(* CODESYS project ApatitKLK1400v5-31.project
   Company: CKA
   Title: Apatit KLK 1400
   Author: Stanislav
   Version: 0.0.0.26

Project tree, tasks and I/O mapping:
  MyController : TM241CE40T/U, Schneider Electric, order no. TM241CE40T/U, version 4.0.6.18
    application Application
      task MAST (cyclic, interval 20 ms, priority 15, watchdog 100 ms x 1) calls Alarm, Operations, Indication, FC, Encoder, LevelSensors, HMI
      task Network (cyclic, interval t#10ms, priority 31) calls nothing
      program Encoder [LD]
      global variables GVL
      program Alarm [LD]
      Symbols
      global variables PersistentVars
      program Operations [LD]
      program Indication [LD]
      program FC [LD]
      program LevelSensors [LD]
      program HMI [LD]
    DI : Digital Inputs, Schneider Electric, version 4.0.6.18
        settings: IOs Usage = 3
        input  idwDI_IDW0 : DWORD  // IDW0
        input  PositionEncoderA : BOOL  // IDW0.I0
        input  PositionEncoderB : BOOL  // IDW0.I1
        input  DKS : BOOL  // IDW0.I2
        input  FaultDKSLA : BOOL  // IDW0.I3
        input  FaultDKSLB : BOOL  // IDW0.I4
        input  FaultDKODriverDrum : BOOL  // IDW0.I5
        input  FaultDKOTensionDrum : BOOL  // IDW0.I6
        input  FaultATVA : BOOL  // IDW0.I7
        input  FaultATVB : BOOL  // IDW0.I8
        input  FrontEndPosition : BOOL  // IDW0.I9
        input  RearEndPosition : BOOL  // IDW0.I10
        input  EmergencyStop : BOOL  // IDW0.I11
        input  FaultTempDriverDrum : BOOL  // IDW0.I12
        input  FaultTempTensionDrum : BOOL  // IDW0.I13
        input  FaultTempSensorBreak : BOOL  // IDW0.I14
        input  PermissionGranted : BOOL  // IDW0.I15
        input  InputModeBeltLocal : BOOL  // IDW0.I16
        input  InputModeBeltAuto : BOOL  // IDW0.I17
        input  InputModeMoveLocal : BOOL  // IDW0.I18
        input  InputModeMoveAuto : BOOL  // IDW0.I19
        input  BeltRemoteForward : BOOL  // IDW0.I20
        input  BeltRemoteReverse : BOOL  // IDW0.I21
        input  BeltRemoteStop : BOOL  // IDW0.I22
        input  MoveRemoteForward : BOOL  // IDW0.I23
        input  ibDI_IB1 : BYTE  // IB1
    DQ : Digital Outputs, Schneider Electric, version 4.0.6.18
        output BeltRunForward : BOOL  // QW0.Q0
        output BeltRunReverse : BOOL  // QW0.Q1
        output MovingForward : BOOL  // QW0.Q2
        output MovingBackward : BOOL  // QW0.Q3
        output IndicationFrontEndPosition : BOOL  // QW0.Q4
        output IndicationRearEndPosition : BOOL  // QW0.Q5
        output StatusReady : BOOL  // QW0.Q6
        output StatusFault : BOOL  // QW0.Q7
        output IndicationModeAutoBelt : BOOL  // QW0.Q8
        output IndicationModeAutoMove : BOOL  // QW0.Q9
        output IndicationFCatSetpoint : BOOL  // QW0.Q10
        output AlarmSignalDevice : BOOL  // QW0.Q11
        output Reserve1 : BOOL  // QW0.Q12
        output Reserve2 : BOOL  // QW0.Q13
        output Reserve3 : BOOL  // QW0.Q14
        output Reserve4 : BOOL  // QW0.Q15
        output qbDQ_QB1 : BYTE  // QB1
        unmapped channels: QW0
    Counters : Counters, Schneider Electric, version 4.0.6.18
        settings: Instance name = 'HscMainDualPhase_0'; B input History = 'old=-1 new=1'; A input History = 'old=-1 new=0'; Temporary Instance name = 'HscMainDualPhase_0'
    Pulse_Generators : Pulse Generators, Schneider Electric, version 4.0.6.18
    Cartridge_1 : Cartridge, Schneider Electric, version 4.0.6.18
    Cartridge_2 : Cartridge, Schneider Electric, version 4.0.6.18
    IO_Bus : IO bus - TM3, Schneider Electric, version 4.0.6.18
      Module_1 : TM3DI16/G, Schneider Electric, order no. TM3DI16/G, version 1.0.1.4
          input  iwModule_1_IW0 : WORD  // IW0
          input  MoveRemoteBackward : BOOL  // IW0.I0
          input  MoveRemoteStop : BOOL  // IW0.I1
          input  AcknowledgmentRemoteAndLocal : BOOL  // IW0.I2
          input  BeltLocalForward : BOOL  // IW0.I3
          input  BeltLocalReverse : BOOL  // IW0.I4
          input  BeltLocalStop : BOOL  // IW0.I5
          input  MoveLocalForward : BOOL  // IW0.I6
          input  MoveLocalBackward : BOOL  // IW0.I7
          input  MoveLocalStop : BOOL  // IW0.I8
          input  BeltAutoForward : BOOL  // IW0.I9
          input  BeltAutoReverse : BOOL  // IW0.I10
          input  MoveAutoForward : BOOL  // IW0.I11
          input  MoveAutoBackward : BOOL  // IW0.I12
          input  FaultPowerSupply : BOOL  // IW0.I13
          input  FaultM1 : BOOL  // IW0.I14
          input  FaultM2M3 : BOOL  // IW0.I15
      Module_2 : TM3AI2H/G, Schneider Electric, order no. TM3AI2H/G, version 1.0.0.17
          settings: KPI Configuration.KPI Configuration[0] = 35; KPI Configuration.KPI Configuration[1] = 35; KPI Configuration.KPI Configuration[2] = 60; KPI Configuration.KPI Configuration[3] = 15; KPI Configuration.KPI Configuration[4] = 60; KPI Configuration.KPI Configuration[5] = 15; KPI Configuration.KPI Configuration[6] = 32; KPI Configuration.KPI Configuration[7] = 78; KPI Configuration.KPI Configuration[8] = 32; KPI Configuration.KPI Configuration[9] = 78
          input  iiModule_2_IW0 : INT  // IW0
          input  iiModule_2_IW1 : INT  // IW1
          input  ibModule_2_IBStatusIW0 : BYTE  // IBStatusIW0
          input  ibModule_2_IBStatusIW1 : BYTE  // IBStatusIW1
    COM_Bus : COM bus, Schneider Electric, version 4.0.6.18
      TM4ES4 : TM4ES4, Schneider Electric, order no. TM4ES4, version 1.0.0.10
          settings: IPAddress = [192, 168, 201, 103]; SubnetMask = [255, 255, 255, 0]; WebServer = FALSE; FTP Server = FALSE; SoMachine Protocol = TRUE; Modbus Server = TRUE; NetManage Protocol = TRUE; SNMP protocol = TRUE; Enable Routing = TRUE; WebVisu protocol = TRUE
    Ethernet_1 : Ethernet Network, Schneider Electric, version 4.0.6.18
        settings: IPAddress = [192, 168, 200, 101]; SubnetMask = [255, 255, 255, 0]; DeviceName = 'PLCKLK1400'; WebServer = TRUE; FTP Server = TRUE; SoMachine Protocol = TRUE; Modbus Server = TRUE; NetManage Protocol = TRUE; SNMP protocol = TRUE; WebVisu protocol = TRUE; DHCP Server Active = TRUE
      Industrial_Ethernet_Manager : Industrial Ethernet Manager, Schneider Electric, version 1.0.12.21
          settings: BinaryFileSize = 396; Dhcps Host 0.Client Mac Address = [16#0, 16#0, 16#0, 16#0, 16#0]; Dhcps Host 0.Client Device Name = 'ATV340_1'; Dhcps Host 0.Client IP Address = [192, 168, 200, 102]; Dhcps Host 0.Network Mask = [255, 255, 255, 0]; Dhcps Host 0.Default Gateway = [192, 168, 200, 101]; Dhcps Host 1.Client Mac Address = [16#0, 16#0, 16#0, 16#0, 16#0]; Dhcps Host 2.Client Mac Address = [16#0, 16#0, 16#0, 16#0, 16#0]; Dhcps Host 3.Client Mac Address = [16#0, 16#0, 16#0, 16#0, 16#0]; Dhcps Host 4.Client Mac Address = [16#0, 16#0, 16#0, 16#0, 16#0]; Dhcps Host 5.Client Mac Address = [16#0, 16#0, 16#0, 16#0, 16#0]; Dhcps Host 6.Client Mac Address = [16#0, 16#0, 16#0, 16#0, 16#0]; Dhcps Host 7.Client Mac Address = [16#0, 16#0, 16#0, 16#0, 16#0]; Dhcps Host 8.Client Mac Address = [16#0, 16#0, 16#0, 16#0, 16#0]; Dhcps Host 9.Client Mac Address = [16#0, 16#0, 16#0, 16#0, 16#0]; Dhcps Host 10.Client Mac Address = [16#0, 16#0, 16#0, 16#0, 16#0]; Dhcps Host 11.Client Mac Address = [16#0, 16#0, 16#0, 16#0, 16#0]; Dhcps Host 12.Client Mac Address = [16#0, 16#0, 16#0, 16#0, 16#0]; Dhcps Host 13.Client Mac Address = [16#0, 16#0, 16#0, 16#0, 16#0]; Dhcps Host 14.Client Mac Address = [16#0, 16#0, 16#0, 16#0, 16#0]; Dhcps Host 15.Client Mac Address = [16#0, 16#0, 16#0, 16#0, 16#0]; Dhcps Host 16.Client Mac Address = [16#0, 16#0, 16#0, 16#0, 16#0]; Dhcps Host 17.Client Mac Address = [16#0, 16#0, 16#0, 16#0, 16#0]; Dhcps Host 18.Client Mac Address = [16#0, 16#0, 16#0, 16#0, 16#0]; Dhcps Host 19.Client Mac Address = [16#0, 16#0, 16#0, 16#0, 16#0]; Dhcps Host 20.Client Mac Address = [16#0, 16#0, 16#0, 16#0, 16#0]; Dhcps Host 21.Client Mac Address = [16#0, 16#0, 16#0, 16#0, 16#0]; Dhcps Host 22.Client Mac Address = [16#0, 16#0, 16#0, 16#0, 16#0]; Dhcps Host 23.Client Mac Address = [16#0, 16#0, 16#0, 16#0, 16#0]; Dhcps Host 24.Client Mac Address = [16#0, 16#0, 16#0, 16#0, 16#0]; Dhcps Host 25.Client Mac Address = [16#0, 16#0, 16#0, 16#0, 16#0]; Dhcps Host 26.Client Mac Address = [16#0, 16#0, 16#0, 16#0, 16#0]; Dhcps Host 27.Client Mac Address = [16#0, 16#0, 16#0, 16#0, 16#0]; Dhcps Host 28.Client Mac Address = [16#0, 16#0, 16#0, 16#0, 16#0]; Dhcps Host 29.Client Mac Address = [16#0, 16#0, 16#0, 16#0, 16#0]; Dhcps Host 30.Client Mac Address = [16#0, 16#0, 16#0, 16#0, 16#0]; Dhcps Host 31.Client Mac Address = [16#0, 16#0, 16#0, 16#0, 16#0]; Dhcps Host 32.Client Mac Address = [16#0, 16#0, 16#0, 16#0, 16#0]; Dhcps Host 33.Client Mac Address = [16#0, 16#0, 16#0, 16#0, 16#0]; Dhcps Host 34.Client Mac Address = [16#0, 16#0, 16#0, 16#0, 16#0];
            Dhcps Host 35.Client Mac Address = [16#0, 16#0, 16#0, 16#0, 16#0]; Dhcps Host 36.Client Mac Address = [16#0, 16#0, 16#0, 16#0, 16#0]; Dhcps Host 37.Client Mac Address = [16#0, 16#0, 16#0, 16#0, 16#0]; Dhcps Host 38.Client Mac Address = [16#0, 16#0, 16#0, 16#0, 16#0]; Dhcps Host 39.Client Mac Address = [16#0, 16#0, 16#0, 16#0, 16#0]; Dhcps Host 40.Client Mac Address = [16#0, 16#0, 16#0, 16#0, 16#0]; Dhcps Host 41.Client Mac Address = [16#0, 16#0, 16#0, 16#0, 16#0]; Dhcps Host 42.Client Mac Address = [16#0, 16#0, 16#0, 16#0, 16#0]; Dhcps Host 43.Client Mac Address = [16#0, 16#0, 16#0, 16#0, 16#0]; Dhcps Host 44.Client Mac Address = [16#0, 16#0, 16#0, 16#0, 16#0]; Dhcps Host 45.Client Mac Address = [16#0, 16#0, 16#0, 16#0, 16#0]; Dhcps Host 46.Client Mac Address = [16#0, 16#0, 16#0, 16#0, 16#0]; Dhcps Host 47.Client Mac Address = [16#0, 16#0, 16#0, 16#0, 16#0]; Dhcps Host 48.Client Mac Address = [16#0, 16#0, 16#0, 16#0, 16#0]; Dhcps Host 49.Client Mac Address = [16#0, 16#0, 16#0, 16#0, 16#0]; Dhcps Host 50.Client Mac Address = [16#0, 16#0, 16#0, 16#0, 16#0]; Dhcps Host 51.Client Mac Address = [16#0, 16#0, 16#0, 16#0, 16#0]; Dhcps Host 52.Client Mac Address = [16#0, 16#0, 16#0, 16#0, 16#0]; Dhcps Host 53.Client Mac Address = [16#0, 16#0, 16#0, 16#0, 16#0]; Dhcps Host 54.Client Mac Address = [16#0, 16#0, 16#0, 16#0, 16#0]; Dhcps Host 55.Client Mac Address = [16#0, 16#0, 16#0, 16#0, 16#0]; Dhcps Host 56.Client Mac Address = [16#0, 16#0, 16#0, 16#0, 16#0]; Dhcps Host 57.Client Mac Address = [16#0, 16#0, 16#0, 16#0, 16#0]; Dhcps Host 58.Client Mac Address = [16#0, 16#0, 16#0, 16#0, 16#0]; Dhcps Host 59.Client Mac Address = [16#0, 16#0, 16#0, 16#0, 16#0]; Dhcps Host 60.Client Mac Address = [16#0, 16#0, 16#0, 16#0, 16#0]; Dhcps Host 61.Client Mac Address = [16#0, 16#0, 16#0, 16#0, 16#0]; Dhcps Host 62.Client Mac Address = [16#0, 16#0, 16#0, 16#0, 16#0]; Dhcps Host 63.Client Mac Address = [16#0, 16#0, 16#0, 16#0, 16#0]; Dhcps Host 64.Client Mac Address = [16#0, 16#0, 16#0, 16#0, 16#0]; Dhcps Host 65.Client Mac Address = [16#0, 16#0, 16#0, 16#0, 16#0]; Dhcps Host 66.Client Mac Address = [16#0, 16#0, 16#0, 16#0, 16#0]; Dhcps Host 67.Client Mac Address = [16#0, 16#0, 16#0, 16#0, 16#0]; Dhcps Host 68.Client Mac Address = [16#0, 16#0, 16#0, 16#0, 16#0]; Dhcps Host 69.Client Mac Address = [16#0, 16#0, 16#0, 16#0, 16#0]; Dhcps Host 70.Client Mac Address = [16#0, 16#0, 16#0, 16#0, 16#0]; Dhcps Host 71.Client Mac Address = [16#0, 16#0, 16#0, 16#0, 16#0]; Dhcps Host 72.Client Mac Address = [16#0, 16#0, 16#0, 16#0, 16#0]; Dhcps Host 73.Client Mac Address = [16#0, 16#0, 16#0, 16#0, 16#0]; Dhcps Host 74.Client Mac Address = [16#0, 16#0, 16#0, 16#0, 16#0];
            Dhcps Host 75.Client Mac Address = [16#0, 16#0, 16#0, 16#0, 16#0]; Dhcps Host 76.Client Mac Address = [16#0, 16#0, 16#0, 16#0, 16#0]; Dhcps Host 77.Client Mac Address = [16#0, 16#0, 16#0, 16#0, 16#0]; Dhcps Host 78.Client Mac Address = [16#0, 16#0, 16#0, 16#0, 16#0]; Dhcps Host 79.Client Mac Address = [16#0, 16#0, 16#0, 16#0, 16#0]; Dhcps Host 80.Client Mac Address = [16#0, 16#0, 16#0, 16#0, 16#0]; Dhcps Host 81.Client Mac Address = [16#0, 16#0, 16#0, 16#0, 16#0]; Dhcps Host 82.Client Mac Address = [16#0, 16#0, 16#0, 16#0, 16#0]; Dhcps Host 83.Client Mac Address = [16#0, 16#0, 16#0, 16#0, 16#0]; Dhcps Host 84.Client Mac Address = [16#0, 16#0, 16#0, 16#0, 16#0]; Dhcps Host 85.Client Mac Address = [16#0, 16#0, 16#0, 16#0, 16#0]; Dhcps Host 86.Client Mac Address = [16#0, 16#0, 16#0, 16#0, 16#0]; Dhcps Host 87.Client Mac Address = [16#0, 16#0, 16#0, 16#0, 16#0]; Dhcps Host 88.Client Mac Address = [16#0, 16#0, 16#0, 16#0, 16#0]; Dhcps Host 89.Client Mac Address = [16#0, 16#0, 16#0, 16#0, 16#0]; Dhcps Host 90.Client Mac Address = [16#0, 16#0, 16#0, 16#0, 16#0]; Dhcps Host 91.Client Mac Address = [16#0, 16#0, 16#0, 16#0, 16#0]; Dhcps Host 92.Client Mac Address = [16#0, 16#0, 16#0, 16#0, 16#0]; Dhcps Host 93.Client Mac Address = [16#0, 16#0, 16#0, 16#0, 16#0]; Dhcps Host 94.Client Mac Address = [16#0, 16#0, 16#0, 16#0, 16#0]; Dhcps Host 95.Client Mac Address = [16#0, 16#0, 16#0, 16#0, 16#0]; Dhcps Host 96.Client Mac Address = [16#0, 16#0, 16#0, 16#0, 16#0]; Dhcps Host 97.Client Mac Address = [16#0, 16#0, 16#0, 16#0, 16#0]; Dhcps Host 98.Client Mac Address = [16#0, 16#0, 16#0, 16#0, 16#0]; Dhcps Host 99.Client Mac Address = [16#0, 16#0, 16#0, 16#0, 16#0]; Dhcps Host 100.Client Mac Address = [16#0, 16#0, 16#0, 16#0, 16#0]; Dhcps Host 101.Client Mac Address = [16#0, 16#0, 16#0, 16#0, 16#0]; Dhcps Host 102.Client Mac Address = [16#0, 16#0, 16#0, 16#0, 16#0]; Dhcps Host 103.Client Mac Address = [16#0, 16#0, 16#0, 16#0, 16#0]; Dhcps Host 104.Client Mac Address = [16#0, 16#0, 16#0, 16#0, 16#0]; Dhcps Host 105.Client Mac Address = [16#0, 16#0, 16#0, 16#0, 16#0]; Dhcps Host 106.Client Mac Address = [16#0, 16#0, 16#0, 16#0, 16#0]; Dhcps Host 107.Client Mac Address = [16#0, 16#0, 16#0, 16#0, 16#0]; Dhcps Host 108.Client Mac Address = [16#0, 16#0, 16#0, 16#0, 16#0]; Dhcps Host 109.Client Mac Address = [16#0, 16#0, 16#0, 16#0, 16#0]; Dhcps Host 110.Client Mac Address = [16#0, 16#0, 16#0, 16#0, 16#0]; Dhcps Host 111.Client Mac Address = [16#0, 16#0, 16#0, 16#0, 16#0]; Dhcps Host 112.Client Mac Address = [16#0, 16#0, 16#0, 16#0, 16#0]; Dhcps Host 113.Client Mac Address = [16#0, 16#0, 16#0, 16#0, 16#0]; Dhcps Host 114.Client Mac Address = [16#0, 16#0, 16#0, 16#0, 16#0];
            Dhcps Host 115.Client Mac Address = [16#0, 16#0, 16#0, 16#0, 16#0]; Dhcps Host 116.Client Mac Address = [16#0, 16#0, 16#0, 16#0, 16#0]; Dhcps Host 117.Client Mac Address = [16#0, 16#0, 16#0, 16#0, 16#0]; Dhcps Host 118.Client Mac Address = [16#0, 16#0, 16#0, 16#0, 16#0]; Dhcps Host 119.Client Mac Address = [16#0, 16#0, 16#0, 16#0, 16#0]; Dhcps Host 120.Client Mac Address = [16#0, 16#0, 16#0, 16#0, 16#0]; Dhcps Host 121.Client Mac Address = [16#0, 16#0, 16#0, 16#0, 16#0]; Dhcps Host 122.Client Mac Address = [16#0, 16#0, 16#0, 16#0, 16#0]; Dhcps Host 123.Client Mac Address = [16#0, 16#0, 16#0, 16#0, 16#0]; Dhcps Host 124.Client Mac Address = [16#0, 16#0, 16#0, 16#0, 16#0]; Dhcps Host 125.Client Mac Address = [16#0, 16#0, 16#0, 16#0, 16#0]; Dhcps Host 126.Client Mac Address = [16#0, 16#0, 16#0, 16#0, 16#0]; Dhcps Host 127.Client Mac Address = [16#0, 16#0, 16#0, 16#0, 16#0]; Dhcps Host 128.Client Mac Address = [16#0, 16#0, 16#0, 16#0, 16#0]; serialized Values = 235c3cdb-0ed9-49ff-9223-9c00a6bcd6bc=0|
          unmapped channels: Global Status, Healthbit 0, Healthbit 1, Healthbit 2, Healthbit 3
        ATV340_1 : Altivar 340, Schneider Electric, order no. 340, version 1.0.12.0
            settings: Default Unit-ID = 248; IPAddress = [192, 168, 200, 102]; ATV340 channel.Channel ID = 0; ATV340 channel.Read Offset = 16#0000; ATV340 channel.Write Offset = 16#0000
            input  Statusword : WORD  // Statusword
            input  Actualspeed : WORD  // Output speed
            input  MotorCurrent : WORD  // InputWord 3
            input  MotorFrequency : WORD  // InputWord 4
            input  MotorVoltage : WORD  // InputWord 5
            input  DriveState : WORD  // InputWord 6
            input  MalfunctionCode : WORD  // InputWord 7
            input  LastError : WORD  // InputWord 8
            input  FaultNumber : WORD  // InputWord 9
            input  ActualError : WORD  // InputWord 10
            input  MotorCurrent2 : WORD  // InputWord 11
            input  StateWord : WORD  // InputWord 12
            input  ETIStateWord : WORD  // InputWord 13
            input  StatusWord2 : WORD  // InputWord 14
            output Controlword : WORD  // Control word
            output SpeedReference : WORD  // Speed reference
            unmapped channels: InputWord 15, InputWord 16, InputWord 17, InputWord 18, InputWord 19, InputWord 20, InputWord 21, InputWord 22, InputWord 23, InputWord 24, InputWord 25, InputWord 26, InputWord 27, InputWord 28, InputWord 29, InputWord 30, InputWord 31, InputWord 32, OutputWord 3, OutputWord 4, OutputWord 5, OutputWord 6, OutputWord 7, OutputWord 8, OutputWord 9, OutputWord 10, OutputWord 11, OutputWord 12, OutputWord 13, OutputWord 14, OutputWord 15, OutputWord 16, OutputWord 17, OutputWord 18, OutputWord 19, OutputWord 20, OutputWord 21, OutputWord 22, OutputWord 23, OutputWord 24,
              OutputWord 25, OutputWord 26, OutputWord 27, OutputWord 28, OutputWord 29, OutputWord 30, OutputWord 31, OutputWord 32
    Serial_Line_1 : Serial line, Schneider Electric, version 4.0.6.18
    Serial_Line_2 : Serial line, Schneider Electric, version 4.0.6.18
      Modbus_Manager : Modbus Manager, Schneider Electric, version 4.0.0.2
  text list GlobalTextList
*)

// MyController/Application/GVL
VAR_GLOBAL
	
	FlagFaultCommon 			AT %MX0.0 : BOOL;
	FaultGroupUniversal 		AT %MX0.1 : BOOL;
	FaultGroupBelt 				AT %MX0.2 : BOOL;
	FaultGroupMove 				AT %MX0.3 : BOOL;
	FlagFaultLowSpeed			AT %MX0.4 : BOOL;
	FlagFaultDKSLA				AT %MX0.5 : BOOL;
	FlagFaultDKSLB				AT %MX0.6 : BOOL;
	FlagFaultDKODriverDrum		AT %MX0.7 : BOOL;
	FlagFaultDKOTensionDrum		AT %MX1.0 : BOOL;
	FlagFaultATVA				AT %MX1.1 : BOOL;
	FlagFaultATVB				AT %MX1.2 : BOOL;
	FlagEmergencyStop			AT %MX1.3 : BOOL;
	FlagFaultTempDriverDrum		AT %MX1.4 : BOOL;
	FlagFaultTempTensionDrum	AT %MX1.5 : BOOL;
	FlagFaultTempSensorBreak	AT %MX1.6 : BOOL;	
	FlagFaultPowerSupply		AT %MX1.7 : BOOL;
	FlagFaultM1					AT %MX2.0 : BOOL;
	FlagFaultM2M3				AT %MX2.1 : BOOL;
	
	CurrentStateBeltFWD			AT %MX2.2 : BOOL;
	CurrentStateBeltREV			AT %MX2.3 : BOOL;
	CurrentStateMoveFWD			AT %MX2.4 : BOOL;
	CurrentStateMoveBWD 		AT %MX2.5 : BOOL;
	
	HMIFrontendPosition			AT %MX2.6 : BOOL;
	HMIRearendPosition			AT %MX2.7 : BOOL;
	HMIReady					AT %MX3.0 : BOOL;
		
	DKSPauseGlobal 				: TIME;
	PrestartBeltPause1 			: TIME := TIME#10S0MS;
	PrestartBeltPause2 			: TIME := TIME#30S0MS;
	PrestartBeltPause3 			: TIME := T#30S;
	PrestartMovePause 			: TIME := T#10S;
	DirectionChangeBeltPause 	: TIME := T#10S;
	DirectionChangeMovePause 	: TIME := T#10S;	

	ServicePrestartBeltPause1 			: TIME;
	ServicePrestartBeltPause2 			: TIME;
	ServicePrestartBeltPause3 			: TIME;
	ServicePrestartMovePause 			: TIME;
	ServiceDirectionChangeBeltPause 	: TIME;
	ServiceDirectionChangeMovePause 	: TIME;
	
	Level1Normal 				AT %MD11 : REAL;
	Level2Normal 				AT %MD12 : REAL;
	
	Position 					AT %MD13 : REAL;
	
	FCParameter1				AT %MW32 : WORD;
	FCParameter2				AT %MW33 : WORD;
	FCParameter3				AT %MW34 : WORD;
	FCParameter4				AT %MW35 : WORD;
	FCParameter5				AT %MW36 : WORD;
	FCParameter6				AT %MW37 : WORD;
	FCParameter7				AT %MW38 : WORD;
	FCParameter8				AT %MW39 : WORD;
	FCParameter9				AT %MW40 : WORD;
	FCParameter10				AT %MW41 : WORD;
	FCParameter11				AT %MW42 : WORD;
	FCParameter12				AT %MW43 : WORD;
	FCParameter13				AT %MW44 : WORD;
	FCParameter14				AT %MW45 : WORD;
	
	Level1Real : REAL;
	Level2Real : REAL;
		
	Level1Error : BOOL;
	Level2Error : BOOL;
	
	FaultReset: BOOL;
	
	FlagPrestartSignalBeltFWD: BOOL;
	FlagPrestartSignalBeltREV: BOOL;
	FlagPrestartSignalMoveFWD: BOOL;
	FlagPrestartSignalMoveBWD: BOOL;
	
	ModeBeltLocal: BOOL;
	ModeBeltRemote: BOOL;
	ModeBeltAuto: BOOL;
	ModeMoveLocal: BOOL;
	ModeMoveRemote: BOOL;
	ModeMoveAuto: BOOL;
	
	TagBeltRunning: BOOL;
	
	TONPrestartBeltPause1: TON;
	TONPrestartBeltPause2: TON;
	TONPrestartBeltPause3: TON;
	TONPrestartMovePause: TON;
	
	AcknowledgmentAuto 		AT %MX92.0: BOOL;
	
	Blinker: BOOL;
	DKSPauseInms: TIME;
	FaultAcknowledged: BOOL;
	
	TurnOnDKS: BOOL;
		
	TONDKSPrestartPause: TON;
	TONAlarmService1: TIME;
	TONFaultM1: TON;
	TONAlarmService2: TIME;
	TONFaultM2M3: TON;
	TONAlarmService3: TIME;
	TONMeander1: TON;
	TONAlarmService4: TIME;
	TONMeander2: TON;
	TONAlarmService5: TIME;
	
	TONBootInputFilter: TON;
	TONDirectionChangeBelt1: TON;
	TONDirectionChangeBelt2: TON;
	TONDirectionChangeMove1: TON;
	TONDirectionChangeMove2: TON;
	
	TONOperationsService0: TIME;
	TONOperationsService1: TIME;
	TONOperationsService2: TIME;
	TONOperationsService3: TIME;
	TONOperationsService4: TIME;
	TONOperationsService5: TIME;
	TONOperationsService6: TIME;
	TONOperationsService7: TIME;
	TONOperationsService8: TIME;
	
	HSCEnable: BOOL;
	HSCPreset: BOOL;
	EncoderEnable: BOOL;
	EncoderPreset: BOOL;
	
	EncoderValueReal: REAL;

	StatusWordAsBits: WORD_AS_BIT;
END_VAR
VAR_GLOBAL CONSTANT
	AlwaysTRUE: BOOL := TRUE;
END_VAR
VAR_GLOBAL RETAIN
	EncoderValue: DINT;
	EncoderValueBackup: DINT;
	
	HMIDKSPauseGlobal 			AT %MW2 : INT;
	HMIPrestartBeltPause1 		AT %MW3 : INT;
	HMIPrestartBeltPause2 		AT %MW4 : INT;
	HMIPrestartBeltPause3 		AT %MW5 : INT;
	HMIPrestartMovePause 		AT %MW6 : INT;
	HMIDirectionChangeBeltPause AT %MW7 : INT;
	HMIDirectionChangeMovePause AT %MW8 : INT;
	
	SpeedLocal 					AT %MW9 : INT;
	SpeedASU 					AT %MW10 : INT;

	EncoderImpulseWeight 		AT %MD6 : REAL;
	Level1min 					AT %MD7 : REAL;
	Level1max 					AT %MD8 : REAL;
	Level2min 					AT %MD9 : REAL;
	Level2max 					AT %MD10 : REAL;
	
	PositionFront 				AT %MD14 : DINT;
	PositionEnd 				AT %MD15 : DINT;
	
	LowSpeedLimit				AT %MD24 : REAL;
	DKSImpulseWeight			AT %MD25 : REAL;
	DKSMeasuredSpeed			AT %MD26 : REAL;
END_VAR

// MyController/Application/PersistentVars
VAR_GLOBAL PERSISTENT RETAIN
	
AlarmFrequency: TIME := T#1S;
	
END_VAR

// MyController/Application/Alarm
PROGRAM Alarm
VAR
	FlagStartCounter: BOOL;
	DKSCounterTimer: TON;
	TONAlarmService6: TIME;
	
	DKSSumImpulses: REAL;
	DKSCTU: CTU;
	DKSBuffer: REAL;
END_VAR
VAR // added by the converter: edge detectors and wires of the graphical bodies
    _w1, _w2 : BOOL;
END_VAR

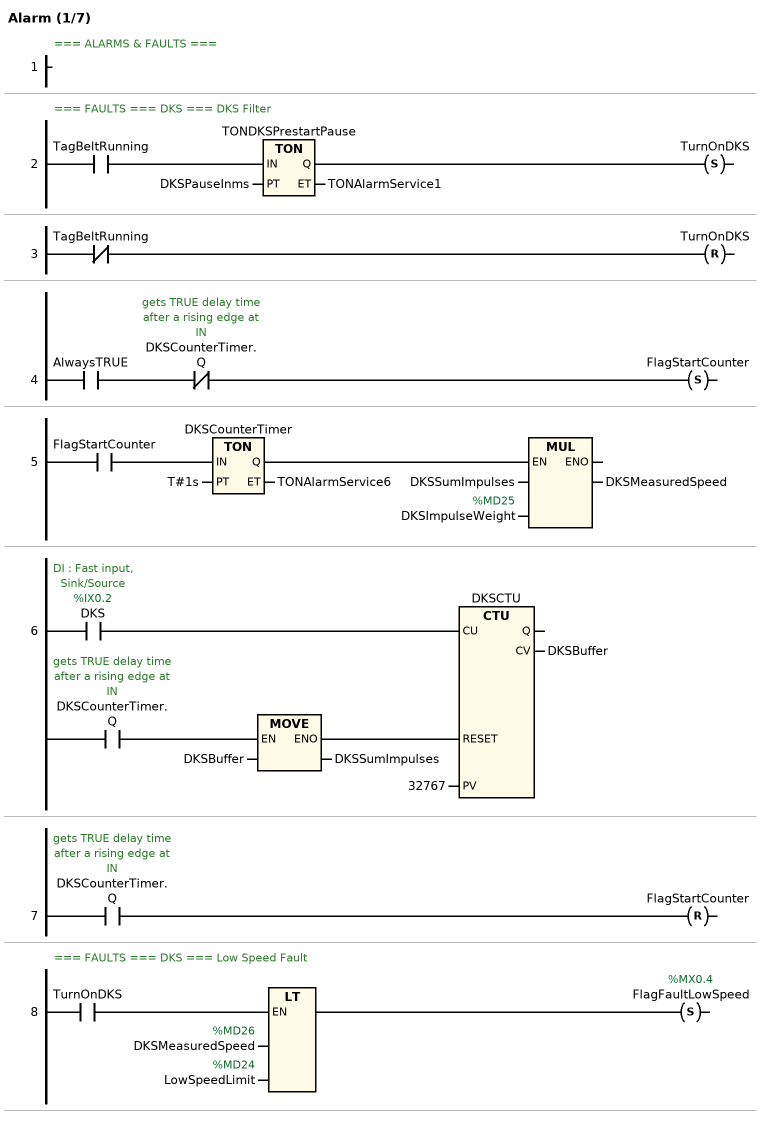
// NETWORK 1
// === ALARMS & FAULTS ===

// NETWORK 2
// === FAULTS === DKS === DKS Filter
TONDKSPrestartPause(IN := TagBeltRunning, PT := DKSPauseInms, ET => TONAlarmService1); // TON
TurnOnDKS S= TONDKSPrestartPause.Q;

// NETWORK 3
TurnOnDKS R= NOT TagBeltRunning;

// NETWORK 4
//   DKSCounterTimer.Q: gets TRUE delay time after a rising edge at IN
FlagStartCounter S= AlwaysTRUE AND NOT DKSCounterTimer.Q;

// NETWORK 5
//   DKSImpulseWeight: AT %MD25
//   DKSMeasuredSpeed: AT %MD26
DKSCounterTimer(IN := FlagStartCounter, PT := T#1s, ET => TONAlarmService6); // TON
IF DKSCounterTimer.Q THEN DKSMeasuredSpeed := DKSSumImpulses * DKSImpulseWeight; END_IF

// NETWORK 6
//   DKS: DI : Fast input, Sink/Source | AT %IX0.2
//   DKSCounterTimer.Q: gets TRUE delay time after a rising edge at IN
_w1 := DKSCounterTimer.Q;
IF _w1 THEN DKSSumImpulses := DKSBuffer; END_IF
DKSCTU(CU := DKS, RESET := _w1, PV := 32767, CV => DKSBuffer); // CTU

// NETWORK 7
//   DKSCounterTimer.Q: gets TRUE delay time after a rising edge at IN
FlagStartCounter R= DKSCounterTimer.Q;

// NETWORK 8
// === FAULTS === DKS === Low Speed Fault
//   DKSMeasuredSpeed: AT %MD26
//   LowSpeedLimit: AT %MD24
//   FlagFaultLowSpeed: AT %MX0.4
FlagFaultLowSpeed S= TurnOnDKS AND DKSMeasuredSpeed < LowSpeedLimit;

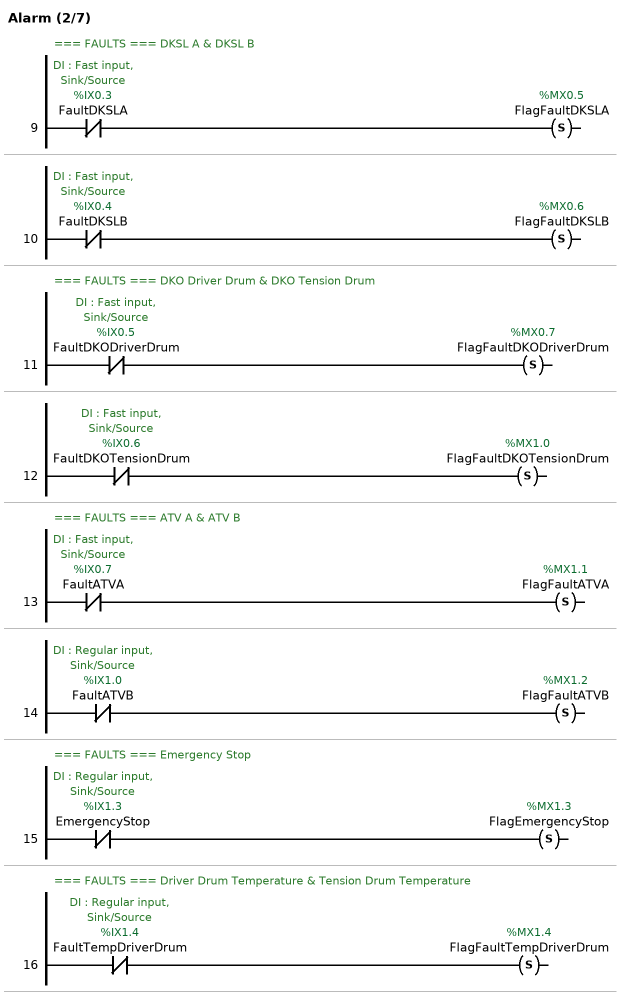
// NETWORK 9
// === FAULTS === DKSL A & DKSL B
//   FaultDKSLA: DI : Fast input, Sink/Source | AT %IX0.3
//   FlagFaultDKSLA: AT %MX0.5
FlagFaultDKSLA S= NOT FaultDKSLA;

// NETWORK 10
//   FaultDKSLB: DI : Fast input, Sink/Source | AT %IX0.4
//   FlagFaultDKSLB: AT %MX0.6
FlagFaultDKSLB S= NOT FaultDKSLB;

// NETWORK 11
// === FAULTS === DKO Driver Drum & DKO Tension Drum
//   FaultDKODriverDrum: DI : Fast input, Sink/Source | AT %IX0.5
//   FlagFaultDKODriverDrum: AT %MX0.7
FlagFaultDKODriverDrum S= NOT FaultDKODriverDrum;

// NETWORK 12
//   FaultDKOTensionDrum: DI : Fast input, Sink/Source | AT %IX0.6
//   FlagFaultDKOTensionDrum: AT %MX1.0
FlagFaultDKOTensionDrum S= NOT FaultDKOTensionDrum;

// NETWORK 13
// === FAULTS === ATV A & ATV B
//   FaultATVA: DI : Fast input, Sink/Source | AT %IX0.7
//   FlagFaultATVA: AT %MX1.1
FlagFaultATVA S= NOT FaultATVA;

// NETWORK 14
//   FaultATVB: DI : Regular input, Sink/Source | AT %IX1.0
//   FlagFaultATVB: AT %MX1.2
FlagFaultATVB S= NOT FaultATVB;

// NETWORK 15
// === FAULTS === Emergency Stop
//   EmergencyStop: DI : Regular input, Sink/Source | AT %IX1.3
//   FlagEmergencyStop: AT %MX1.3
FlagEmergencyStop S= NOT EmergencyStop;

// NETWORK 16
// === FAULTS === Driver Drum Temperature & Tension Drum Temperature
//   FaultTempDriverDrum: DI : Regular input, Sink/Source | AT %IX1.4
//   FlagFaultTempDriverDrum: AT %MX1.4
FlagFaultTempDriverDrum S= NOT FaultTempDriverDrum;

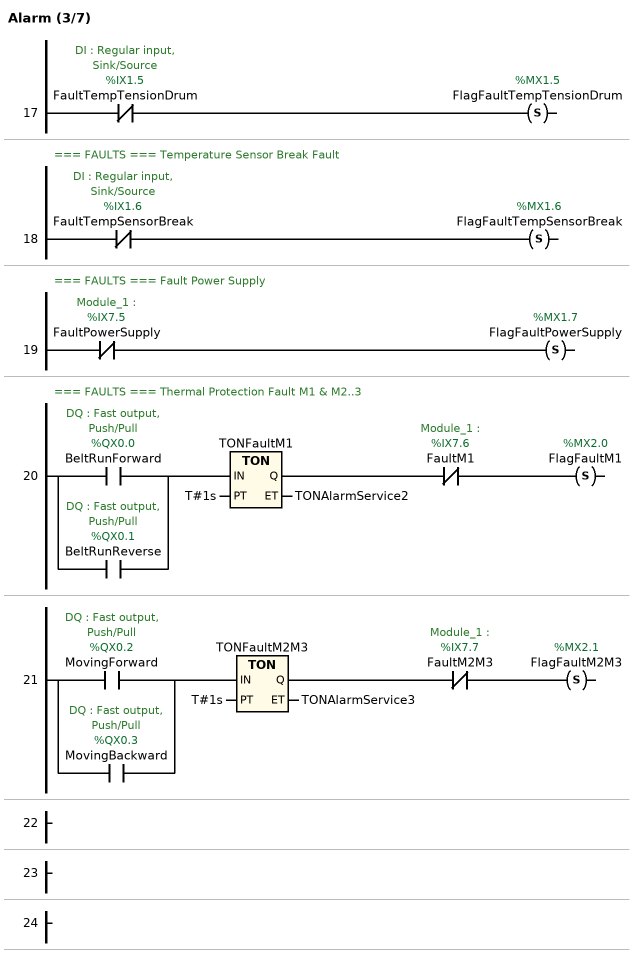
// NETWORK 17
//   FaultTempTensionDrum: DI : Regular input, Sink/Source | AT %IX1.5
//   FlagFaultTempTensionDrum: AT %MX1.5
FlagFaultTempTensionDrum S= NOT FaultTempTensionDrum;

// NETWORK 18
// === FAULTS === Temperature Sensor Break Fault
//   FaultTempSensorBreak: DI : Regular input, Sink/Source | AT %IX1.6
//   FlagFaultTempSensorBreak: AT %MX1.6
FlagFaultTempSensorBreak S= NOT FaultTempSensorBreak;

// NETWORK 19
// === FAULTS === Fault Power Supply
//   FaultPowerSupply: Module_1 : | AT %IX7.5
//   FlagFaultPowerSupply: AT %MX1.7
FlagFaultPowerSupply S= NOT FaultPowerSupply;

// NETWORK 20
// === FAULTS === Thermal Protection Fault M1 & M2..3
//   BeltRunForward: DQ : Fast output, Push/Pull | AT %QX0.0
//   BeltRunReverse: DQ : Fast output, Push/Pull | AT %QX0.1
//   FaultM1: Module_1 : | AT %IX7.6
//   FlagFaultM1: AT %MX2.0
TONFaultM1(IN := BeltRunForward OR BeltRunReverse, PT := T#1s, ET => TONAlarmService2); // TON
FlagFaultM1 S= TONFaultM1.Q AND NOT FaultM1;

// NETWORK 21
//   MovingForward: DQ : Fast output, Push/Pull | AT %QX0.2
//   MovingBackward: DQ : Fast output, Push/Pull | AT %QX0.3
//   FaultM2M3: Module_1 : | AT %IX7.7
//   FlagFaultM2M3: AT %MX2.1
TONFaultM2M3(IN := MovingForward OR MovingBackward, PT := T#1s, ET => TONAlarmService3); // TON
FlagFaultM2M3 S= TONFaultM2M3.Q AND NOT FaultM2M3;

// NETWORK 22

// NETWORK 23

// NETWORK 24

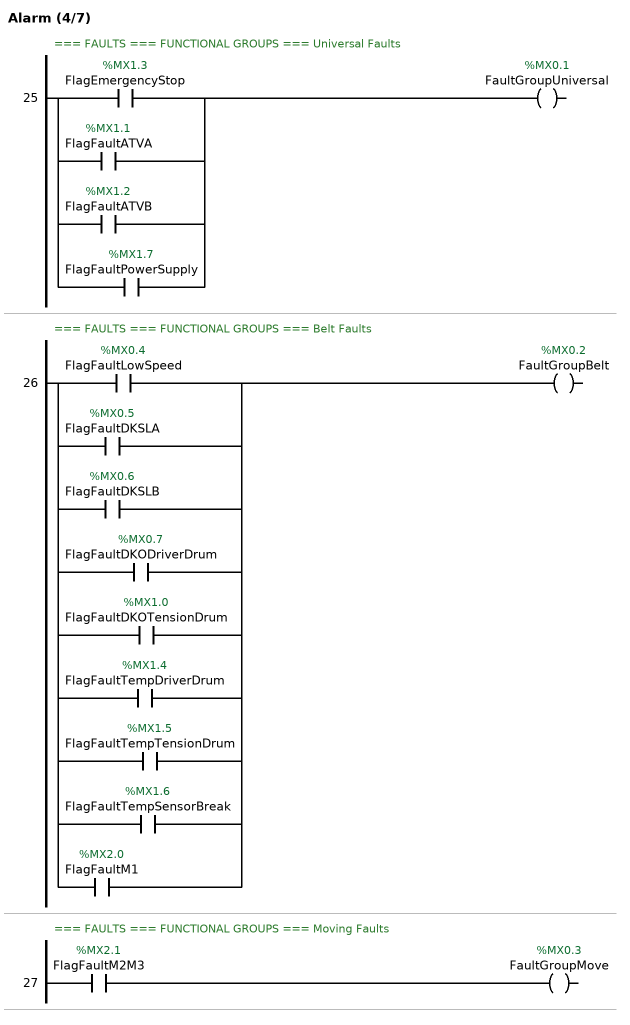
// NETWORK 25
// === FAULTS === FUNCTIONAL GROUPS === Universal Faults
//   FlagEmergencyStop: AT %MX1.3
//   FlagFaultATVA: AT %MX1.1
//   FlagFaultATVB: AT %MX1.2
//   FlagFaultPowerSupply: AT %MX1.7
//   FaultGroupUniversal: AT %MX0.1
FaultGroupUniversal := FlagEmergencyStop OR FlagFaultATVA OR FlagFaultATVB OR FlagFaultPowerSupply;

// NETWORK 26
// === FAULTS === FUNCTIONAL GROUPS === Belt Faults
//   FlagFaultLowSpeed: AT %MX0.4
//   FlagFaultDKSLA: AT %MX0.5
//   FlagFaultDKSLB: AT %MX0.6
//   FlagFaultDKODriverDrum: AT %MX0.7
//   FlagFaultDKOTensionDrum: AT %MX1.0
//   FlagFaultTempDriverDrum: AT %MX1.4
//   FlagFaultTempTensionDrum: AT %MX1.5
//   FlagFaultTempSensorBreak: AT %MX1.6
//   FlagFaultM1: AT %MX2.0
//   FaultGroupBelt: AT %MX0.2
FaultGroupBelt := FlagFaultLowSpeed OR FlagFaultDKSLA OR FlagFaultDKSLB OR FlagFaultDKODriverDrum OR FlagFaultDKOTensionDrum OR FlagFaultTempDriverDrum OR FlagFaultTempTensionDrum OR FlagFaultTempSensorBreak OR FlagFaultM1;

// NETWORK 27
// === FAULTS === FUNCTIONAL GROUPS === Moving Faults
//   FlagFaultM2M3: AT %MX2.1
//   FaultGroupMove: AT %MX0.3
FaultGroupMove := FlagFaultM2M3;

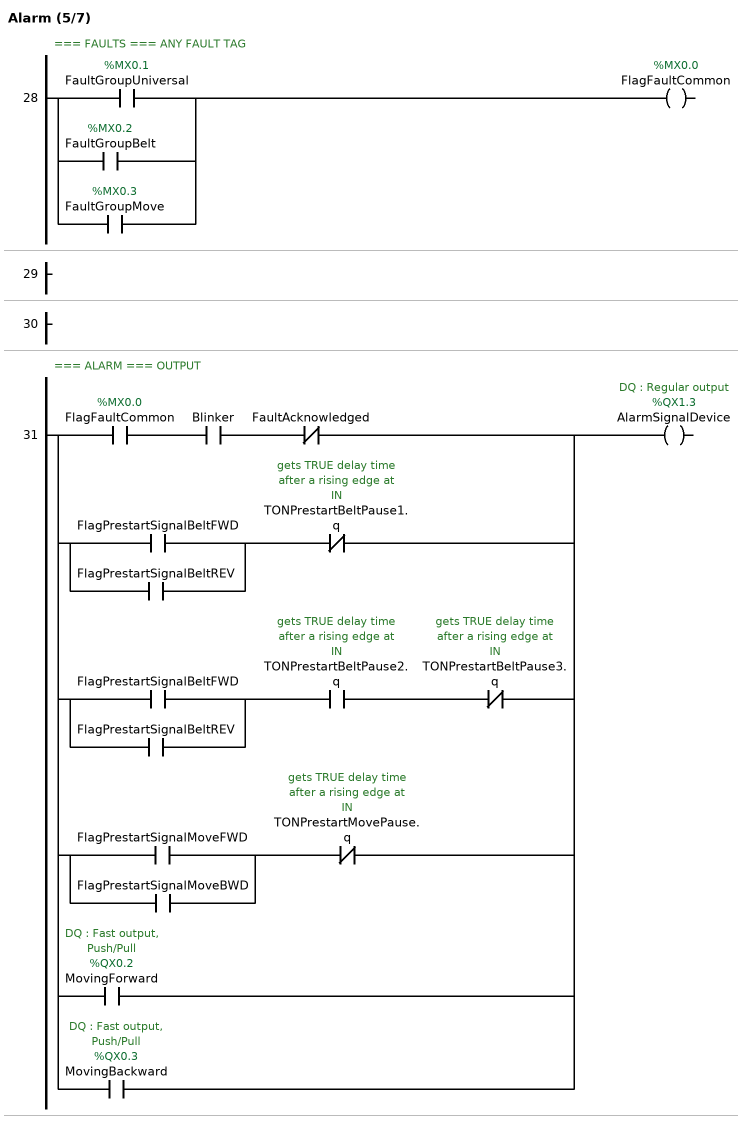
// NETWORK 28
// === FAULTS === ANY FAULT TAG
//   FaultGroupUniversal: AT %MX0.1
//   FaultGroupBelt: AT %MX0.2
//   FaultGroupMove: AT %MX0.3
//   FlagFaultCommon: AT %MX0.0
FlagFaultCommon := FaultGroupUniversal OR FaultGroupBelt OR FaultGroupMove;

// NETWORK 29

// NETWORK 30

// NETWORK 31
// === ALARM === OUTPUT
//   FlagFaultCommon: AT %MX0.0
//   TONPrestartBeltPause1.q: gets TRUE delay time after a rising edge at IN
//   TONPrestartBeltPause2.q: gets TRUE delay time after a rising edge at IN
//   TONPrestartBeltPause3.q: gets TRUE delay time after a rising edge at IN
//   TONPrestartMovePause.q: gets TRUE delay time after a rising edge at IN
//   MovingForward: DQ : Fast output, Push/Pull | AT %QX0.2
//   MovingBackward: DQ : Fast output, Push/Pull | AT %QX0.3
//   AlarmSignalDevice: DQ : Regular output | AT %QX1.3
AlarmSignalDevice := FlagFaultCommon AND Blinker AND NOT FaultAcknowledged OR (FlagPrestartSignalBeltFWD OR FlagPrestartSignalBeltREV) AND NOT TONPrestartBeltPause1.q OR (FlagPrestartSignalBeltFWD OR FlagPrestartSignalBeltREV) AND TONPrestartBeltPause2.q AND NOT TONPrestartBeltPause3.q OR (FlagPrestartSignalMoveFWD OR FlagPrestartSignalMoveBWD) AND NOT TONPrestartMovePause.q OR MovingForward OR MovingBackward;

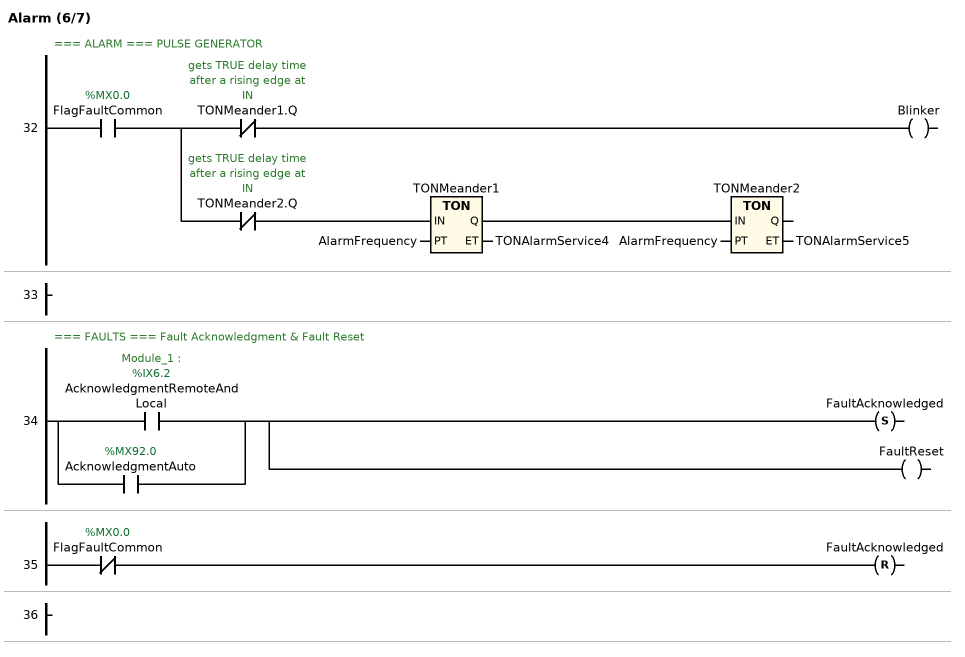
// NETWORK 32
// === ALARM === PULSE GENERATOR
//   FlagFaultCommon: AT %MX0.0
//   TONMeander1.Q: gets TRUE delay time after a rising edge at IN
//   TONMeander2.Q: gets TRUE delay time after a rising edge at IN
Blinker := FlagFaultCommon AND NOT TONMeander1.Q;
TONMeander1(IN := FlagFaultCommon AND NOT TONMeander2.Q, PT := AlarmFrequency, ET => TONAlarmService4); // TON
TONMeander2(IN := TONMeander1.Q, PT := AlarmFrequency, ET => TONAlarmService5); // TON

// NETWORK 33

// NETWORK 34
// === FAULTS === Fault Acknowledgment & Fault Reset
//   AcknowledgmentRemoteAndLocal: Module_1 : | AT %IX6.2
//   AcknowledgmentAuto: AT %MX92.0
_w2 := AcknowledgmentRemoteAndLocal OR AcknowledgmentAuto;
FaultAcknowledged S= _w2;
FaultReset := _w2;

// NETWORK 35
//   FlagFaultCommon: AT %MX0.0
FaultAcknowledged R= NOT FlagFaultCommon;

// NETWORK 36

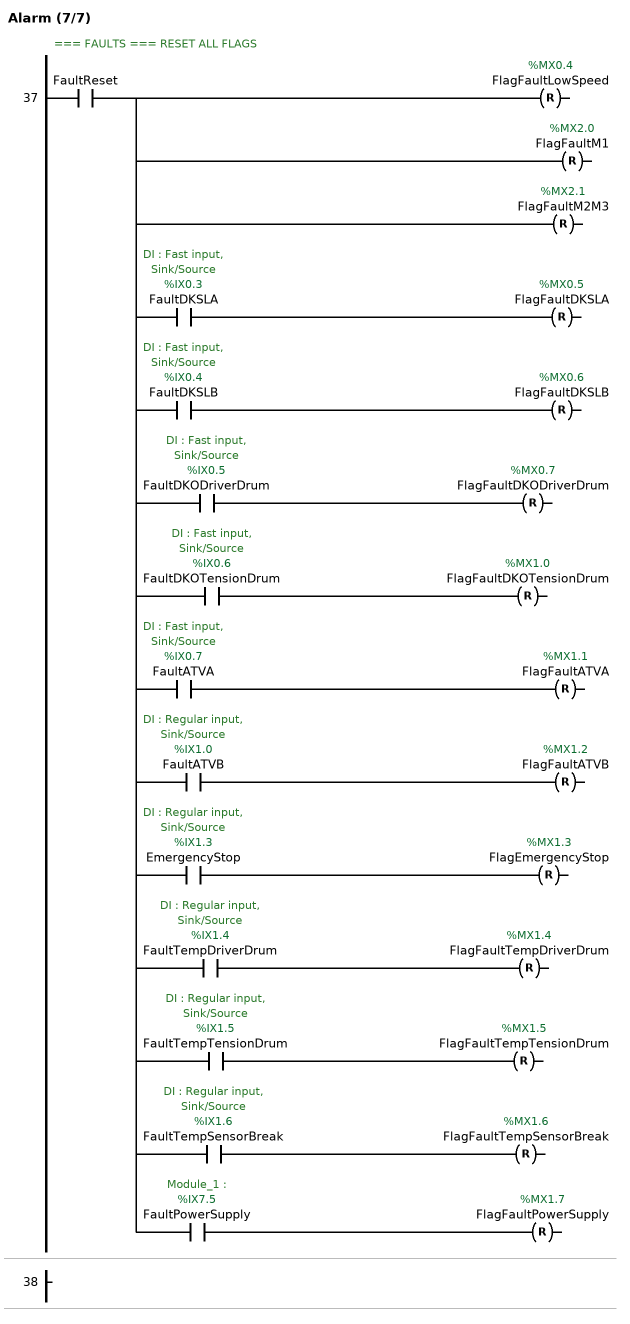
// NETWORK 37
// === FAULTS === RESET ALL FLAGS
//   FlagFaultLowSpeed: AT %MX0.4
//   FlagFaultM1: AT %MX2.0
//   FlagFaultM2M3: AT %MX2.1
//   FaultDKSLA: DI : Fast input, Sink/Source | AT %IX0.3
//   FlagFaultDKSLA: AT %MX0.5
//   FaultDKSLB: DI : Fast input, Sink/Source | AT %IX0.4
//   FlagFaultDKSLB: AT %MX0.6
//   FaultDKODriverDrum: DI : Fast input, Sink/Source | AT %IX0.5
//   FlagFaultDKODriverDrum: AT %MX0.7
//   FaultDKOTensionDrum: DI : Fast input, Sink/Source | AT %IX0.6
//   FlagFaultDKOTensionDrum: AT %MX1.0
//   FaultATVA: DI : Fast input, Sink/Source | AT %IX0.7
//   FlagFaultATVA: AT %MX1.1
//   FaultATVB: DI : Regular input, Sink/Source | AT %IX1.0
//   FlagFaultATVB: AT %MX1.2
//   EmergencyStop: DI : Regular input, Sink/Source | AT %IX1.3
//   FlagEmergencyStop: AT %MX1.3
//   FaultTempDriverDrum: DI : Regular input, Sink/Source | AT %IX1.4
//   FlagFaultTempDriverDrum: AT %MX1.4
//   FaultTempTensionDrum: DI : Regular input, Sink/Source | AT %IX1.5
//   FlagFaultTempTensionDrum: AT %MX1.5
//   FaultTempSensorBreak: DI : Regular input, Sink/Source | AT %IX1.6
//   FlagFaultTempSensorBreak: AT %MX1.6
//   FaultPowerSupply: Module_1 : | AT %IX7.5
//   FlagFaultPowerSupply: AT %MX1.7
FlagFaultLowSpeed R= FaultReset;
FlagFaultM1 R= FaultReset;
FlagFaultM2M3 R= FaultReset;
FlagFaultDKSLA R= FaultReset AND FaultDKSLA;
FlagFaultDKSLB R= FaultReset AND FaultDKSLB;
FlagFaultDKODriverDrum R= FaultReset AND FaultDKODriverDrum;
FlagFaultDKOTensionDrum R= FaultReset AND FaultDKOTensionDrum;
FlagFaultATVA R= FaultReset AND FaultATVA;
FlagFaultATVB R= FaultReset AND FaultATVB;
FlagEmergencyStop R= FaultReset AND EmergencyStop;
FlagFaultTempDriverDrum R= FaultReset AND FaultTempDriverDrum;
FlagFaultTempTensionDrum R= FaultReset AND FaultTempTensionDrum;
FlagFaultTempSensorBreak R= FaultReset AND FaultTempSensorBreak;
FlagFaultPowerSupply R= FaultReset AND FaultPowerSupply;

// NETWORK 38

END_PROGRAM

// MyController/Application/Operations
PROGRAM Operations
VAR

END_VAR
VAR // added by the converter: edge detectors and wires of the graphical bodies
    _rt1, _rt2, _rt3, _rt4, _rt5, _rt6, _rt7, _rt8 : R_TRIG;
    _ft1, _ft2, _ft3, _ft4, _ft5, _ft6, _ft7, _ft8, _ft9, _ft10 : F_TRIG;
    _w1, _w2, _w3, _w4 : BOOL;
END_VAR

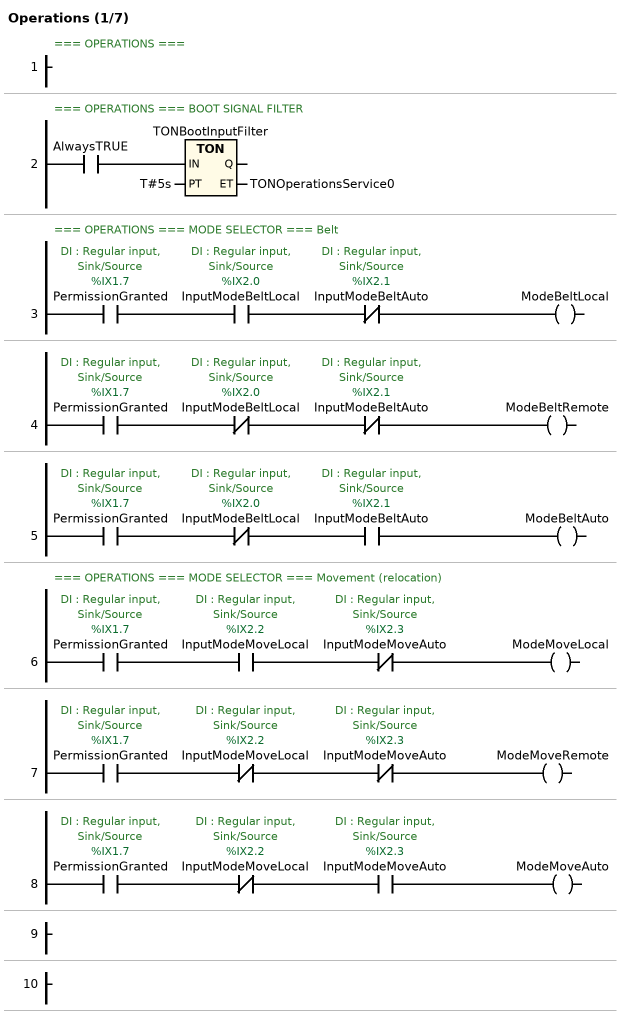
// NETWORK 1
// === OPERATIONS ===

// NETWORK 2
// === OPERATIONS === BOOT SIGNAL FILTER
TONBootInputFilter(IN := AlwaysTRUE, PT := T#5s, ET => TONOperationsService0); // TON

// NETWORK 3
// === OPERATIONS === MODE SELECTOR === Belt
//   PermissionGranted: DI : Regular input, Sink/Source | AT %IX1.7
//   InputModeBeltLocal: DI : Regular input, Sink/Source | AT %IX2.0
//   InputModeBeltAuto: DI : Regular input, Sink/Source | AT %IX2.1
ModeBeltLocal := PermissionGranted AND InputModeBeltLocal AND NOT InputModeBeltAuto;

// NETWORK 4
//   PermissionGranted: DI : Regular input, Sink/Source | AT %IX1.7
//   InputModeBeltLocal: DI : Regular input, Sink/Source | AT %IX2.0
//   InputModeBeltAuto: DI : Regular input, Sink/Source | AT %IX2.1
ModeBeltRemote := PermissionGranted AND NOT InputModeBeltLocal AND NOT InputModeBeltAuto;

// NETWORK 5
//   PermissionGranted: DI : Regular input, Sink/Source | AT %IX1.7
//   InputModeBeltLocal: DI : Regular input, Sink/Source | AT %IX2.0
//   InputModeBeltAuto: DI : Regular input, Sink/Source | AT %IX2.1
ModeBeltAuto := PermissionGranted AND NOT InputModeBeltLocal AND InputModeBeltAuto;

// NETWORK 6
// === OPERATIONS === MODE SELECTOR === Movement (relocation)
//   PermissionGranted: DI : Regular input, Sink/Source | AT %IX1.7
//   InputModeMoveLocal: DI : Regular input, Sink/Source | AT %IX2.2
//   InputModeMoveAuto: DI : Regular input, Sink/Source | AT %IX2.3
ModeMoveLocal := PermissionGranted AND InputModeMoveLocal AND NOT InputModeMoveAuto;

// NETWORK 7
//   PermissionGranted: DI : Regular input, Sink/Source | AT %IX1.7
//   InputModeMoveLocal: DI : Regular input, Sink/Source | AT %IX2.2
//   InputModeMoveAuto: DI : Regular input, Sink/Source | AT %IX2.3
ModeMoveRemote := PermissionGranted AND NOT InputModeMoveLocal AND NOT InputModeMoveAuto;

// NETWORK 8
//   PermissionGranted: DI : Regular input, Sink/Source | AT %IX1.7
//   InputModeMoveLocal: DI : Regular input, Sink/Source | AT %IX2.2
//   InputModeMoveAuto: DI : Regular input, Sink/Source | AT %IX2.3
ModeMoveAuto := PermissionGranted AND NOT InputModeMoveLocal AND InputModeMoveAuto;

// NETWORK 9

// NETWORK 10

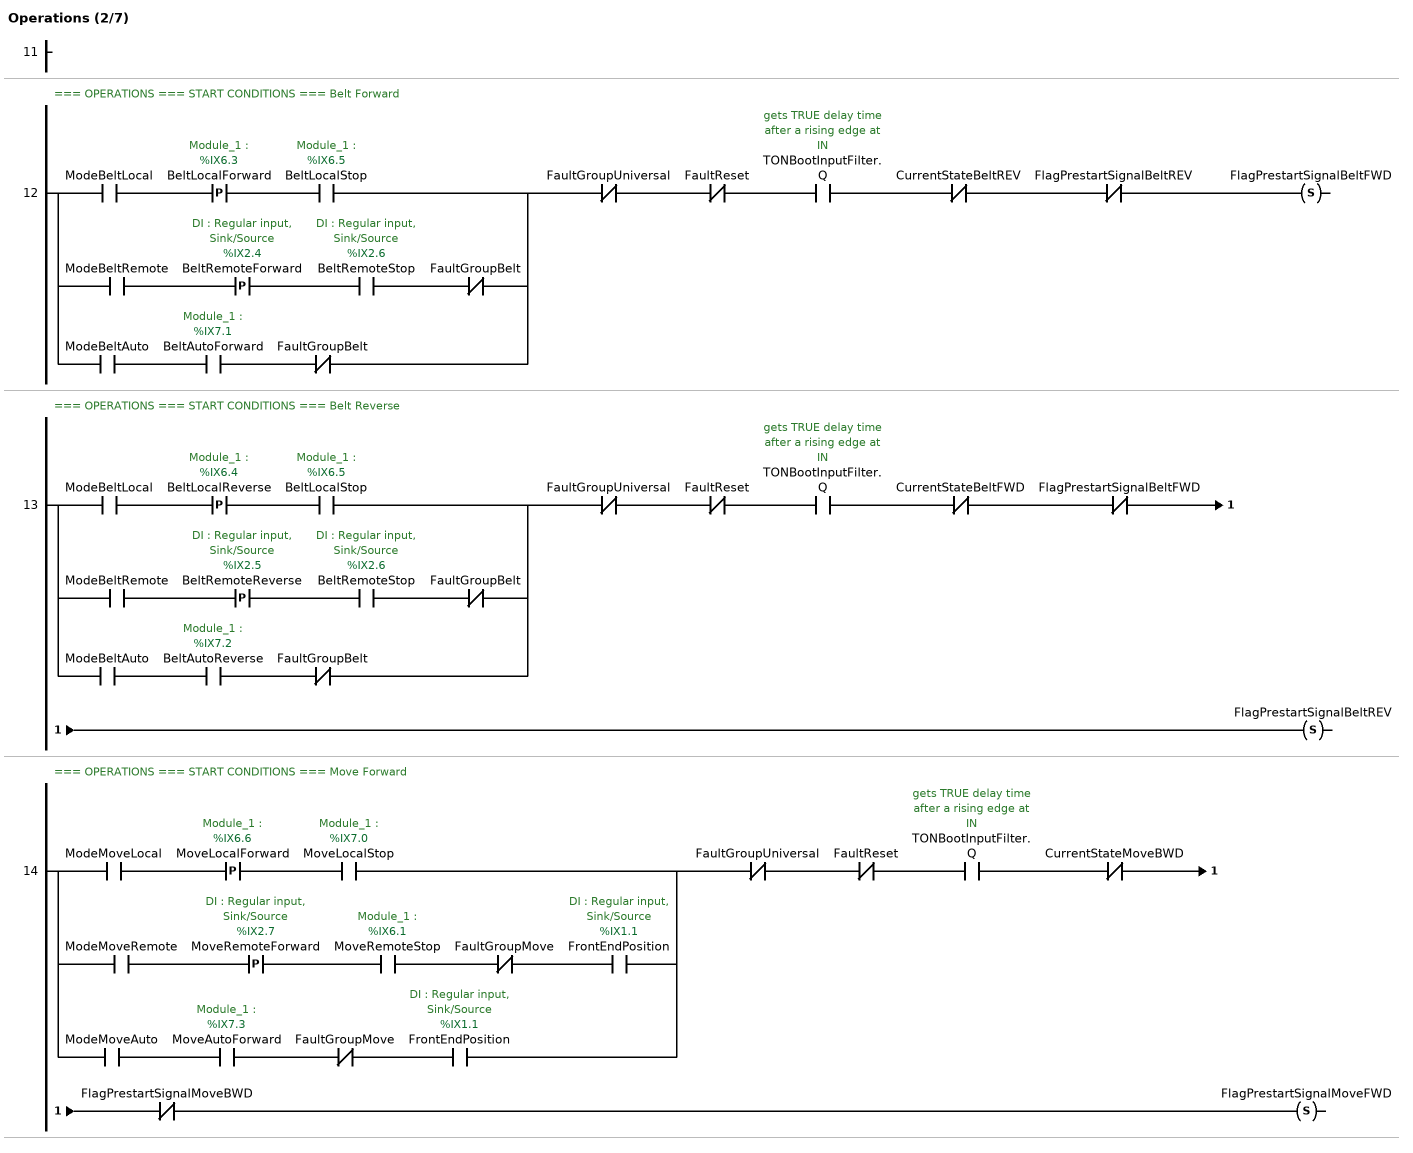
// NETWORK 11

// NETWORK 12
// === OPERATIONS === START CONDITIONS === Belt Forward
//   BeltLocalForward: Module_1 : | AT %IX6.3
//   BeltLocalStop: Module_1 : | AT %IX6.5
//   BeltRemoteForward: DI : Regular input, Sink/Source | AT %IX2.4
//   BeltRemoteStop: DI : Regular input, Sink/Source | AT %IX2.6
//   BeltAutoForward: Module_1 : | AT %IX7.1
//   TONBootInputFilter.Q: gets TRUE delay time after a rising edge at IN
_rt1(CLK := BeltLocalForward);
_rt2(CLK := BeltRemoteForward);
FlagPrestartSignalBeltFWD S= (ModeBeltLocal AND _rt1.Q AND BeltLocalStop OR ModeBeltRemote AND _rt2.Q AND BeltRemoteStop AND NOT FaultGroupBelt OR ModeBeltAuto AND BeltAutoForward AND NOT FaultGroupBelt) AND NOT FaultGroupUniversal AND NOT FaultReset AND TONBootInputFilter.Q AND NOT CurrentStateBeltREV AND NOT FlagPrestartSignalBeltREV;

// NETWORK 13
// === OPERATIONS === START CONDITIONS === Belt Reverse
//   BeltLocalReverse: Module_1 : | AT %IX6.4
//   BeltLocalStop: Module_1 : | AT %IX6.5
//   BeltRemoteReverse: DI : Regular input, Sink/Source | AT %IX2.5
//   BeltRemoteStop: DI : Regular input, Sink/Source | AT %IX2.6
//   BeltAutoReverse: Module_1 : | AT %IX7.2
//   TONBootInputFilter.Q: gets TRUE delay time after a rising edge at IN
_rt3(CLK := BeltLocalReverse);
_rt4(CLK := BeltRemoteReverse);
FlagPrestartSignalBeltREV S= (ModeBeltLocal AND _rt3.Q AND BeltLocalStop OR ModeBeltRemote AND _rt4.Q AND BeltRemoteStop AND NOT FaultGroupBelt OR ModeBeltAuto AND BeltAutoReverse AND NOT FaultGroupBelt) AND NOT FaultGroupUniversal AND NOT FaultReset AND TONBootInputFilter.Q AND NOT CurrentStateBeltFWD AND NOT FlagPrestartSignalBeltFWD;

// NETWORK 14
// === OPERATIONS === START CONDITIONS === Move Forward
//   MoveLocalForward: Module_1 : | AT %IX6.6
//   MoveLocalStop: Module_1 : | AT %IX7.0
//   MoveRemoteForward: DI : Regular input, Sink/Source | AT %IX2.7
//   MoveRemoteStop: Module_1 : | AT %IX6.1
//   FrontEndPosition: DI : Regular input, Sink/Source | AT %IX1.1
//   MoveAutoForward: Module_1 : | AT %IX7.3
//   TONBootInputFilter.Q: gets TRUE delay time after a rising edge at IN
_rt5(CLK := MoveLocalForward);
_rt6(CLK := MoveRemoteForward);
FlagPrestartSignalMoveFWD S= (ModeMoveLocal AND _rt5.Q AND MoveLocalStop OR ModeMoveRemote AND _rt6.Q AND MoveRemoteStop AND NOT FaultGroupMove AND FrontEndPosition OR ModeMoveAuto AND MoveAutoForward AND NOT FaultGroupMove AND FrontEndPosition) AND NOT FaultGroupUniversal AND NOT FaultReset AND TONBootInputFilter.Q AND NOT CurrentStateMoveBWD AND NOT FlagPrestartSignalMoveBWD;

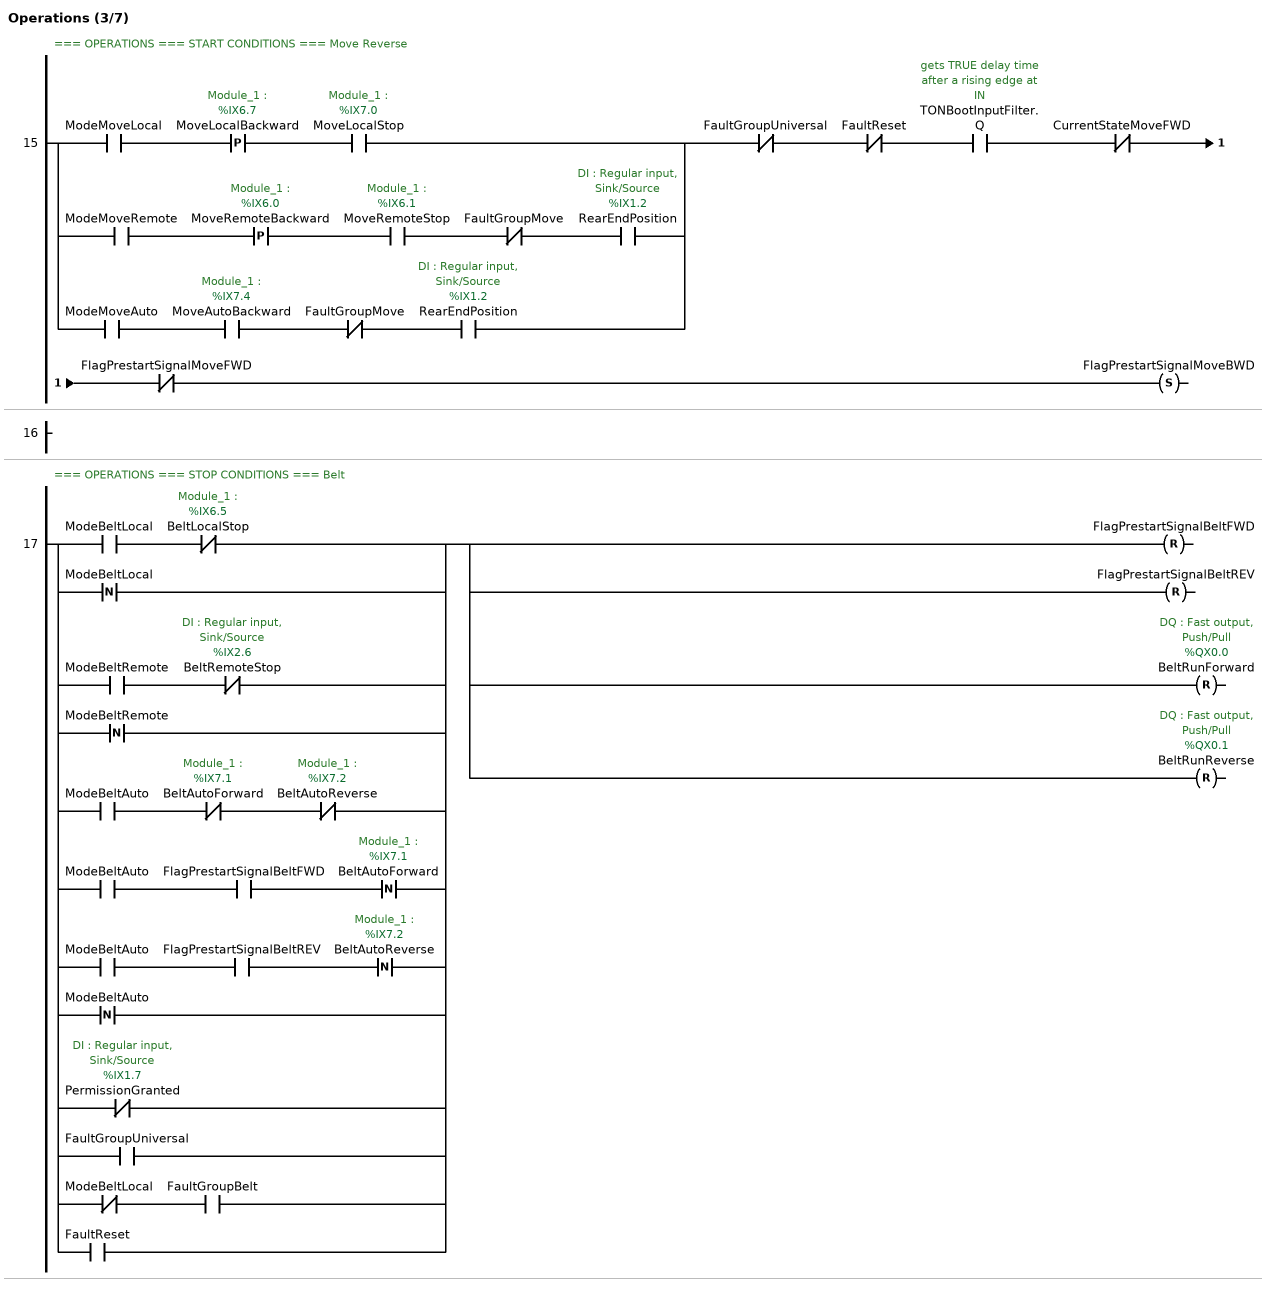
// NETWORK 15
// === OPERATIONS === START CONDITIONS === Move Reverse
//   MoveLocalBackward: Module_1 : | AT %IX6.7
//   MoveLocalStop: Module_1 : | AT %IX7.0
//   MoveRemoteBackward: Module_1 : | AT %IX6.0
//   MoveRemoteStop: Module_1 : | AT %IX6.1
//   RearEndPosition: DI : Regular input, Sink/Source | AT %IX1.2
//   MoveAutoBackward: Module_1 : | AT %IX7.4
//   TONBootInputFilter.Q: gets TRUE delay time after a rising edge at IN
_rt7(CLK := MoveLocalBackward);
_rt8(CLK := MoveRemoteBackward);
FlagPrestartSignalMoveBWD S= (ModeMoveLocal AND _rt7.Q AND MoveLocalStop OR ModeMoveRemote AND _rt8.Q AND MoveRemoteStop AND NOT FaultGroupMove AND RearEndPosition OR ModeMoveAuto AND MoveAutoBackward AND NOT FaultGroupMove AND RearEndPosition) AND NOT FaultGroupUniversal AND NOT FaultReset AND TONBootInputFilter.Q AND NOT CurrentStateMoveFWD AND NOT FlagPrestartSignalMoveFWD;

// NETWORK 16

// NETWORK 17
// === OPERATIONS === STOP CONDITIONS === Belt
//   BeltLocalStop: Module_1 : | AT %IX6.5
//   BeltRemoteStop: DI : Regular input, Sink/Source | AT %IX2.6
//   BeltAutoForward: Module_1 : | AT %IX7.1
//   BeltAutoReverse: Module_1 : | AT %IX7.2
//   PermissionGranted: DI : Regular input, Sink/Source | AT %IX1.7
//   BeltRunForward: DQ : Fast output, Push/Pull | AT %QX0.0
//   BeltRunReverse: DQ : Fast output, Push/Pull | AT %QX0.1
_ft1(CLK := ModeBeltLocal);
_ft2(CLK := ModeBeltRemote);
_ft3(CLK := BeltAutoForward);
_ft4(CLK := BeltAutoReverse);
_ft5(CLK := ModeBeltAuto);
_w1 := ModeBeltLocal AND NOT BeltLocalStop OR _ft1.Q OR ModeBeltRemote AND NOT BeltRemoteStop OR _ft2.Q OR ModeBeltAuto AND NOT BeltAutoForward AND NOT BeltAutoReverse OR ModeBeltAuto AND FlagPrestartSignalBeltFWD AND _ft3.Q OR ModeBeltAuto AND FlagPrestartSignalBeltREV AND _ft4.Q OR _ft5.Q OR NOT PermissionGranted OR FaultGroupUniversal OR NOT ModeBeltLocal AND FaultGroupBelt OR FaultReset;
FlagPrestartSignalBeltFWD R= _w1;
FlagPrestartSignalBeltREV R= _w1;
BeltRunForward R= _w1;
BeltRunReverse R= _w1;

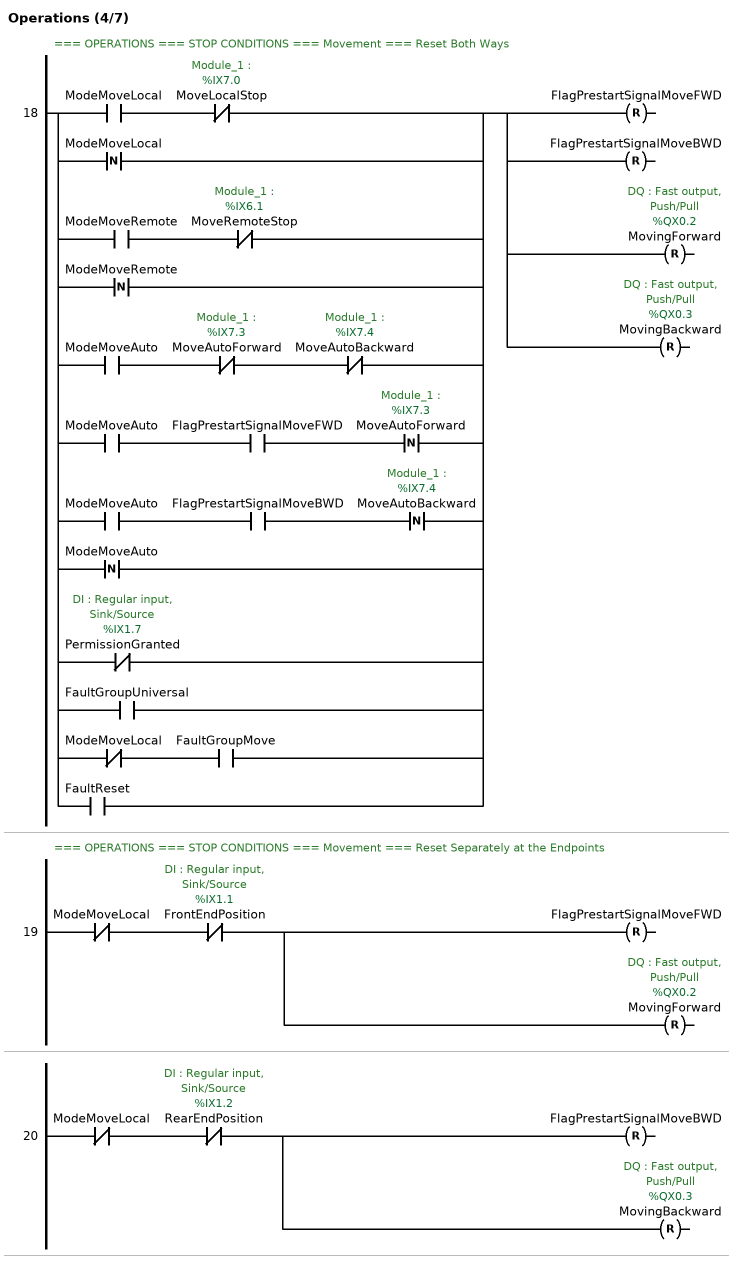
// NETWORK 18
// === OPERATIONS === STOP CONDITIONS === Movement === Reset Both Ways
//   MoveLocalStop: Module_1 : | AT %IX7.0
//   MoveRemoteStop: Module_1 : | AT %IX6.1
//   MoveAutoForward: Module_1 : | AT %IX7.3
//   MoveAutoBackward: Module_1 : | AT %IX7.4
//   PermissionGranted: DI : Regular input, Sink/Source | AT %IX1.7
//   MovingForward: DQ : Fast output, Push/Pull | AT %QX0.2
//   MovingBackward: DQ : Fast output, Push/Pull | AT %QX0.3
_ft6(CLK := ModeMoveLocal);
_ft7(CLK := ModeMoveRemote);
_ft8(CLK := MoveAutoForward);
_ft9(CLK := MoveAutoBackward);
_ft10(CLK := ModeMoveAuto);
_w2 := ModeMoveLocal AND NOT MoveLocalStop OR _ft6.Q OR ModeMoveRemote AND NOT MoveRemoteStop OR _ft7.Q OR ModeMoveAuto AND NOT MoveAutoForward AND NOT MoveAutoBackward OR ModeMoveAuto AND FlagPrestartSignalMoveFWD AND _ft8.Q OR ModeMoveAuto AND FlagPrestartSignalMoveBWD AND _ft9.Q OR _ft10.Q OR NOT PermissionGranted OR FaultGroupUniversal OR NOT ModeMoveLocal AND FaultGroupMove OR FaultReset;
FlagPrestartSignalMoveFWD R= _w2;
FlagPrestartSignalMoveBWD R= _w2;
MovingForward R= _w2;
MovingBackward R= _w2;

// NETWORK 19
// === OPERATIONS === STOP CONDITIONS === Movement === Reset Separately at the Endpoints
//   FrontEndPosition: DI : Regular input, Sink/Source | AT %IX1.1
//   MovingForward: DQ : Fast output, Push/Pull | AT %QX0.2
_w3 := NOT ModeMoveLocal AND NOT FrontEndPosition;
FlagPrestartSignalMoveFWD R= _w3;
MovingForward R= _w3;

// NETWORK 20
//   RearEndPosition: DI : Regular input, Sink/Source | AT %IX1.2
//   MovingBackward: DQ : Fast output, Push/Pull | AT %QX0.3
_w4 := NOT ModeMoveLocal AND NOT RearEndPosition;
FlagPrestartSignalMoveBWD R= _w4;
MovingBackward R= _w4;

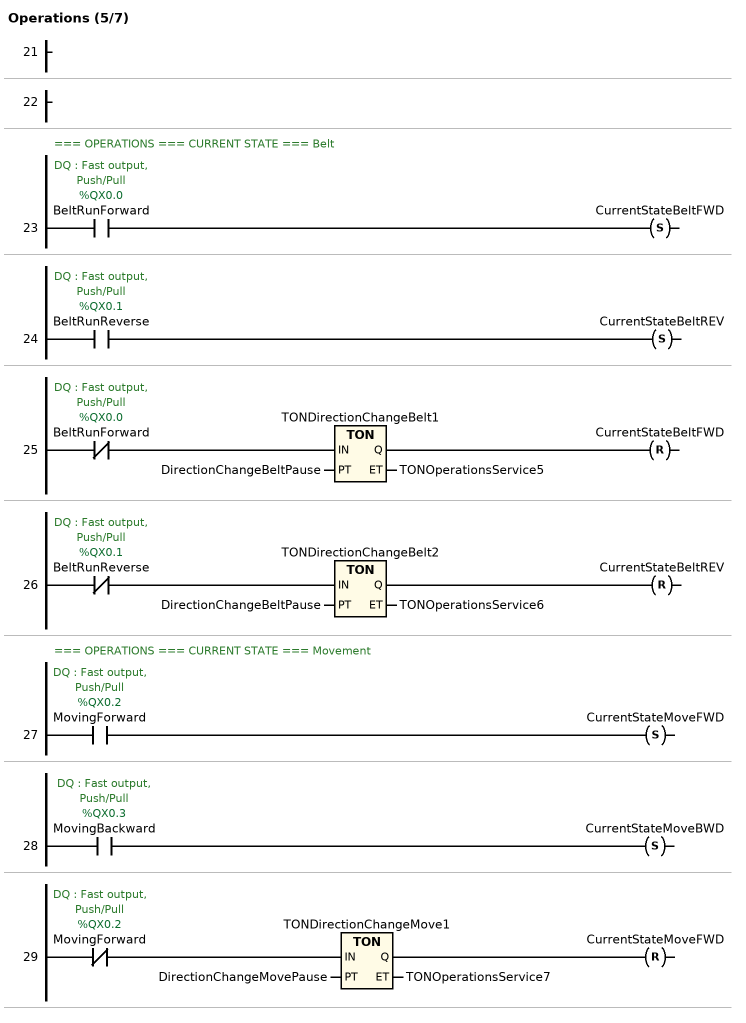
// NETWORK 21

// NETWORK 22

// NETWORK 23
// === OPERATIONS === CURRENT STATE === Belt
//   BeltRunForward: DQ : Fast output, Push/Pull | AT %QX0.0
CurrentStateBeltFWD S= BeltRunForward;

// NETWORK 24
//   BeltRunReverse: DQ : Fast output, Push/Pull | AT %QX0.1
CurrentStateBeltREV S= BeltRunReverse;

// NETWORK 25
//   BeltRunForward: DQ : Fast output, Push/Pull | AT %QX0.0
TONDirectionChangeBelt1(
    IN := NOT BeltRunForward,
    PT := DirectionChangeBeltPause,
    ET => TONOperationsService5); // TON
CurrentStateBeltFWD R= TONDirectionChangeBelt1.Q;

// NETWORK 26
//   BeltRunReverse: DQ : Fast output, Push/Pull | AT %QX0.1
TONDirectionChangeBelt2(
    IN := NOT BeltRunReverse,
    PT := DirectionChangeBeltPause,
    ET => TONOperationsService6); // TON
CurrentStateBeltREV R= TONDirectionChangeBelt2.Q;

// NETWORK 27
// === OPERATIONS === CURRENT STATE === Movement
//   MovingForward: DQ : Fast output, Push/Pull | AT %QX0.2
CurrentStateMoveFWD S= MovingForward;

// NETWORK 28
//   MovingBackward: DQ : Fast output, Push/Pull | AT %QX0.3
CurrentStateMoveBWD S= MovingBackward;

// NETWORK 29
//   MovingForward: DQ : Fast output, Push/Pull | AT %QX0.2
TONDirectionChangeMove1(IN := NOT MovingForward, PT := DirectionChangeMovePause, ET => TONOperationsService7); // TON
CurrentStateMoveFWD R= TONDirectionChangeMove1.Q;

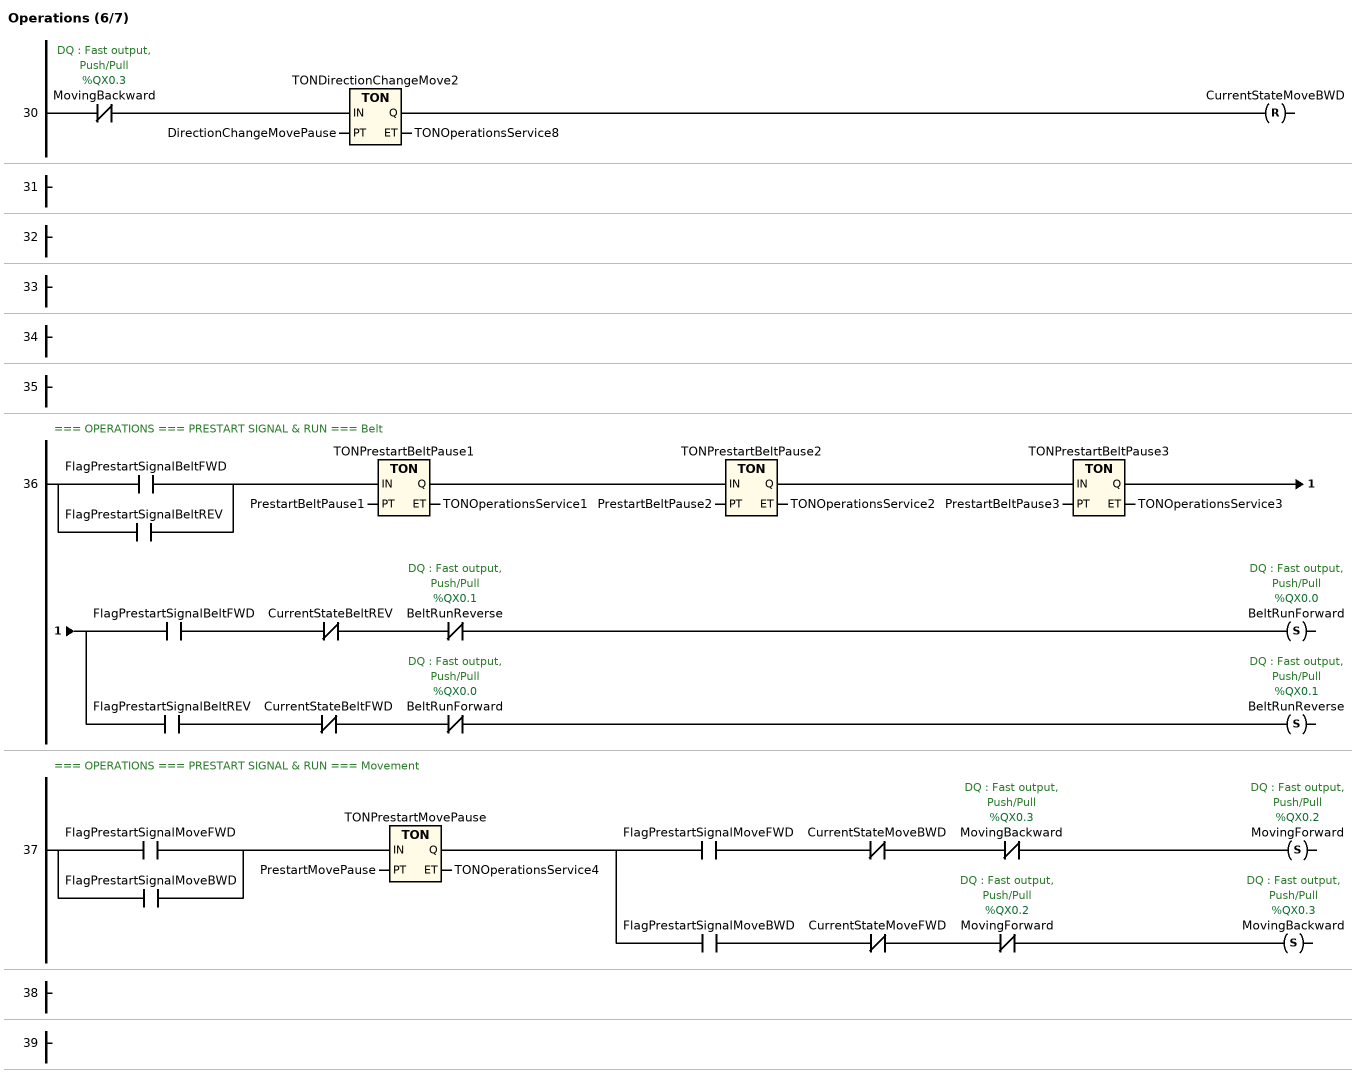
// NETWORK 30
//   MovingBackward: DQ : Fast output, Push/Pull | AT %QX0.3
TONDirectionChangeMove2(
    IN := NOT MovingBackward,
    PT := DirectionChangeMovePause,
    ET => TONOperationsService8); // TON
CurrentStateMoveBWD R= TONDirectionChangeMove2.Q;

// NETWORK 31

// NETWORK 32

// NETWORK 33

// NETWORK 34

// NETWORK 35

// NETWORK 36
// === OPERATIONS === PRESTART SIGNAL & RUN === Belt
//   BeltRunReverse: DQ : Fast output, Push/Pull | AT %QX0.1
//   BeltRunForward: DQ : Fast output, Push/Pull | AT %QX0.0
TONPrestartBeltPause1(
    IN := FlagPrestartSignalBeltFWD OR FlagPrestartSignalBeltREV,
    PT := PrestartBeltPause1,
    ET => TONOperationsService1); // TON
TONPrestartBeltPause2(IN := TONPrestartBeltPause1.Q, PT := PrestartBeltPause2, ET => TONOperationsService2); // TON
TONPrestartBeltPause3(IN := TONPrestartBeltPause2.Q, PT := PrestartBeltPause3, ET => TONOperationsService3); // TON
BeltRunForward S= TONPrestartBeltPause3.Q AND FlagPrestartSignalBeltFWD AND NOT CurrentStateBeltREV AND NOT BeltRunReverse;
BeltRunReverse S= TONPrestartBeltPause3.Q AND FlagPrestartSignalBeltREV AND NOT CurrentStateBeltFWD AND NOT BeltRunForward;

// NETWORK 37
// === OPERATIONS === PRESTART SIGNAL & RUN === Movement
//   MovingBackward: DQ : Fast output, Push/Pull | AT %QX0.3
//   MovingForward: DQ : Fast output, Push/Pull | AT %QX0.2
TONPrestartMovePause(
    IN := FlagPrestartSignalMoveFWD OR FlagPrestartSignalMoveBWD,
    PT := PrestartMovePause,
    ET => TONOperationsService4); // TON
MovingForward S= TONPrestartMovePause.Q AND FlagPrestartSignalMoveFWD AND NOT CurrentStateMoveBWD AND NOT MovingBackward;
MovingBackward S= TONPrestartMovePause.Q AND FlagPrestartSignalMoveBWD AND NOT CurrentStateMoveFWD AND NOT MovingForward;

// NETWORK 38

// NETWORK 39

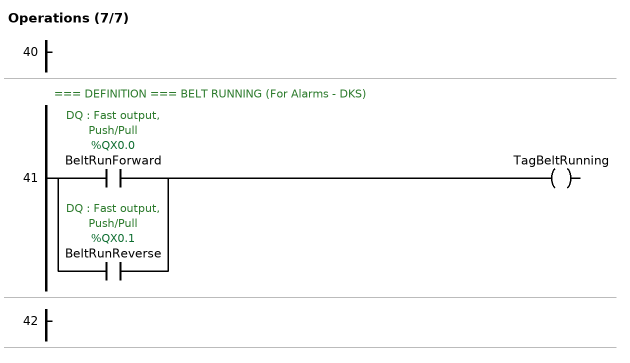
// NETWORK 40

// NETWORK 41
// === DEFINITION === BELT RUNNING (For Alarms - DKS)
//   BeltRunForward: DQ : Fast output, Push/Pull | AT %QX0.0
//   BeltRunReverse: DQ : Fast output, Push/Pull | AT %QX0.1
TagBeltRunning := BeltRunForward OR BeltRunReverse;

// NETWORK 42

END_PROGRAM

// MyController/Application/Indication
PROGRAM Indication
VAR
END_VAR
VAR // added by the converter: edge detectors and wires of the graphical bodies
    _w1, _w2, _w3 : BOOL;
END_VAR

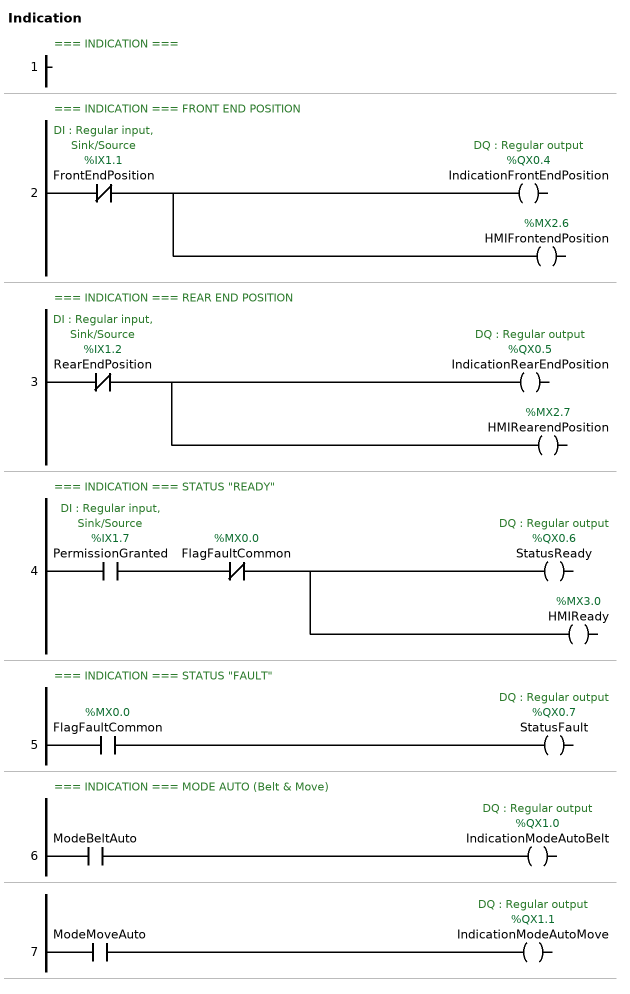
// NETWORK 1
// === INDICATION ===

// NETWORK 2
// === INDICATION === FRONT END POSITION
//   FrontEndPosition: DI : Regular input, Sink/Source | AT %IX1.1
//   IndicationFrontEndPosition: DQ : Regular output | AT %QX0.4
//   HMIFrontendPosition: AT %MX2.6
_w1 := NOT FrontEndPosition;
IndicationFrontEndPosition := _w1;
HMIFrontendPosition := _w1;

// NETWORK 3
// === INDICATION === REAR END POSITION
//   RearEndPosition: DI : Regular input, Sink/Source | AT %IX1.2
//   IndicationRearEndPosition: DQ : Regular output | AT %QX0.5
//   HMIRearendPosition: AT %MX2.7
_w2 := NOT RearEndPosition;
IndicationRearEndPosition := _w2;
HMIRearendPosition := _w2;

// NETWORK 4
// === INDICATION === STATUS "READY"
//   PermissionGranted: DI : Regular input, Sink/Source | AT %IX1.7
//   FlagFaultCommon: AT %MX0.0
//   StatusReady: DQ : Regular output | AT %QX0.6
//   HMIReady: AT %MX3.0
_w3 := PermissionGranted AND NOT FlagFaultCommon;
StatusReady := _w3;
HMIReady := _w3;

// NETWORK 5
// === INDICATION === STATUS "FAULT"
//   FlagFaultCommon: AT %MX0.0
//   StatusFault: DQ : Regular output | AT %QX0.7
StatusFault := FlagFaultCommon;

// NETWORK 6
// === INDICATION === MODE AUTO (Belt & Move)
//   IndicationModeAutoBelt: DQ : Regular output | AT %QX1.0
IndicationModeAutoBelt := ModeBeltAuto;

// NETWORK 7
//   IndicationModeAutoMove: DQ : Regular output | AT %QX1.1
IndicationModeAutoMove := ModeMoveAuto;

END_PROGRAM

// MyController/Application/FC
PROGRAM FC
VAR
	// Function block for I/O device 'ATV340_1'
	fbControl_ATV340_1: GIATV.Control_ATV;
	xCmdEn_ATV340_1: BOOL;
	xCmdKeepOpEn_ATV340_1: BOOL;
	xCmdFwd_ATV340_1: BOOL;
	xCmdRev_ATV340_1: BOOL;
	xCmdQckStop_ATV340_1: BOOL := TRUE;
	xCmdFreeWhl_ATV340_1: BOOL := TRUE;
	xCmdFltRst_ATV340_1: BOOL;
	wSpdRef_ATV340_1: WORD;
	xErrDetected_ATV340_1: BOOL;
	iActualVelo_ATV340_1: INT;
	testWord: WORD;
	SpeedChosen: INT;
	SpeedConverted: INT;
	testBool: BOOL;
	StoppingFlag: BOOL;
	StoppingPause: TON;
	TONPauseService: TIME;
	Statusbit1 : BOOL;
	Statusbit2 : BOOL;
	Statusbit3 : BOOL;
	Statusbit4 : BOOL;
	Statusbit5 : BOOL;
	Statusbit6 : BOOL;
	Statusbit7 : BOOL;
	Statusbit8 : BOOL;
	Statusbit9 : BOOL;
	Statusbit10 : BOOL;
	Statusbit11 : BOOL;
	Statusbit12 : BOOL;
	Statusbit13 : BOOL;
	Statusbit14 : BOOL;
	Statusbit15 : BOOL;
	Statusbit16 : BOOL;

	
END_VAR
VAR // added by the converter: edge detectors and wires of the graphical bodies
    _ft1, _ft2 : F_TRIG;
END_VAR

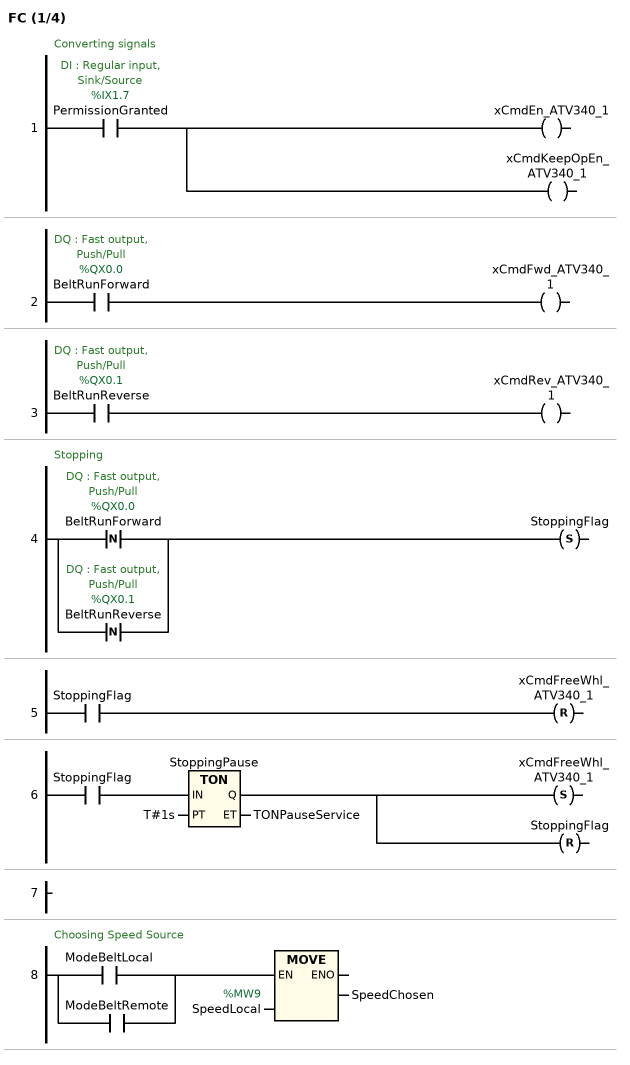
// NETWORK 1
// Converting signals
//   PermissionGranted: DI : Regular input, Sink/Source | AT %IX1.7
xCmdEn_ATV340_1 := PermissionGranted;
xCmdKeepOpEn_ATV340_1 := PermissionGranted;

// NETWORK 2
//   BeltRunForward: DQ : Fast output, Push/Pull | AT %QX0.0
xCmdFwd_ATV340_1 := BeltRunForward;

// NETWORK 3
//   BeltRunReverse: DQ : Fast output, Push/Pull | AT %QX0.1
xCmdRev_ATV340_1 := BeltRunReverse;

// NETWORK 4
// Stopping
//   BeltRunForward: DQ : Fast output, Push/Pull | AT %QX0.0
//   BeltRunReverse: DQ : Fast output, Push/Pull | AT %QX0.1
_ft1(CLK := BeltRunForward);
_ft2(CLK := BeltRunReverse);
StoppingFlag S= _ft1.Q OR _ft2.Q;

// NETWORK 5
xCmdFreeWhl_ATV340_1 R= StoppingFlag;

// NETWORK 6
StoppingPause(IN := StoppingFlag, PT := T#1s, ET => TONPauseService); // TON
xCmdFreeWhl_ATV340_1 S= StoppingPause.Q;
StoppingFlag R= StoppingPause.Q;

// NETWORK 7

// NETWORK 8
// Choosing Speed Source
//   SpeedLocal: AT %MW9
IF ModeBeltLocal OR ModeBeltRemote THEN SpeedChosen := SpeedLocal; END_IF

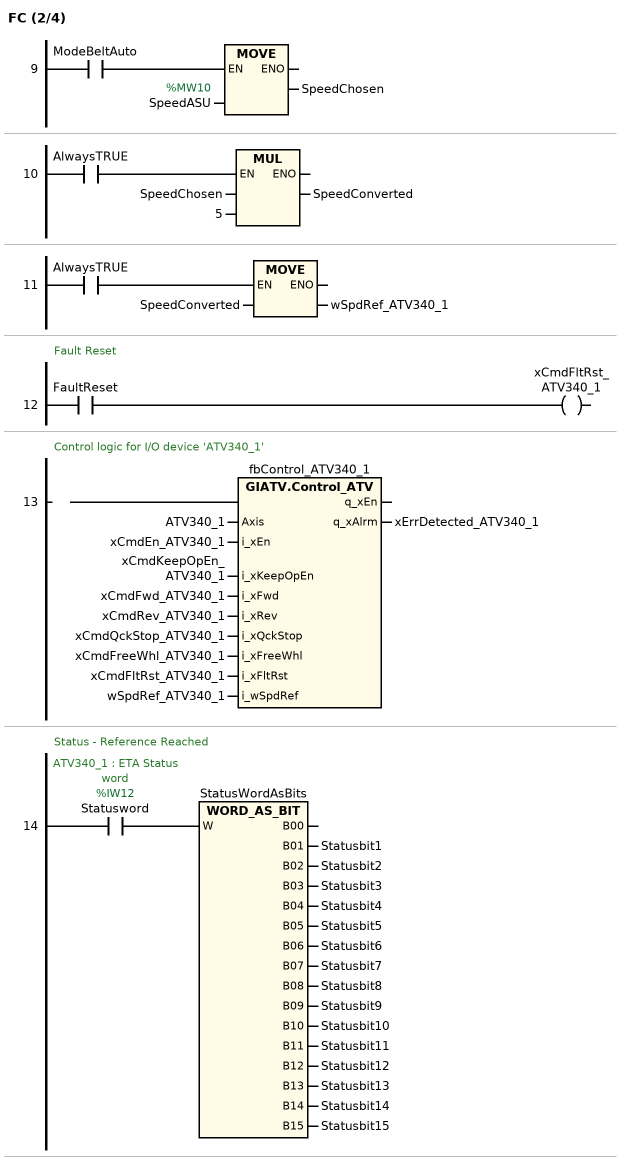
// NETWORK 9
//   SpeedASU: AT %MW10
IF ModeBeltAuto THEN SpeedChosen := SpeedASU; END_IF

// NETWORK 10
IF AlwaysTRUE THEN SpeedConverted := SpeedChosen * 5; END_IF

// NETWORK 11
IF AlwaysTRUE THEN wSpdRef_ATV340_1 := SpeedConverted; END_IF

// NETWORK 12
// Fault Reset
xCmdFltRst_ATV340_1 := FaultReset;

// NETWORK 13
// Control logic for I/O device 'ATV340_1'
//   fbControl_ATV340_1: Function block for I/O device 'ATV340_1'
fbControl_ATV340_1(
    Axis := ATV340_1,
    i_xEn := xCmdEn_ATV340_1,
    i_xKeepOpEn := xCmdKeepOpEn_ATV340_1,
    i_xFwd := xCmdFwd_ATV340_1,
    i_xRev := xCmdRev_ATV340_1,
    i_xQckStop := xCmdQckStop_ATV340_1,
    i_xFreeWhl := xCmdFreeWhl_ATV340_1,
    i_xFltRst := xCmdFltRst_ATV340_1,
    i_wSpdRef := wSpdRef_ATV340_1,
    q_xAlrm => xErrDetected_ATV340_1); // GIATV.Control_ATV

// NETWORK 14
// Status - Reference Reached
//   Statusword: ATV340_1 : ETA Status word | AT %IW12
StatusWordAsBits(
    W := Statusword,
    B01 => Statusbit1,
    B02 => Statusbit2,
    B03 => Statusbit3,
    B04 => Statusbit4,
    B05 => Statusbit5,
    B06 => Statusbit6,
    B07 => Statusbit7,
    B08 => Statusbit8,
    B09 => Statusbit9,
    B10 => Statusbit10,
    B11 => Statusbit11,
    B12 => Statusbit12,
    B13 => Statusbit13,
    B14 => Statusbit14,
    B15 => Statusbit15); // WORD_AS_BIT

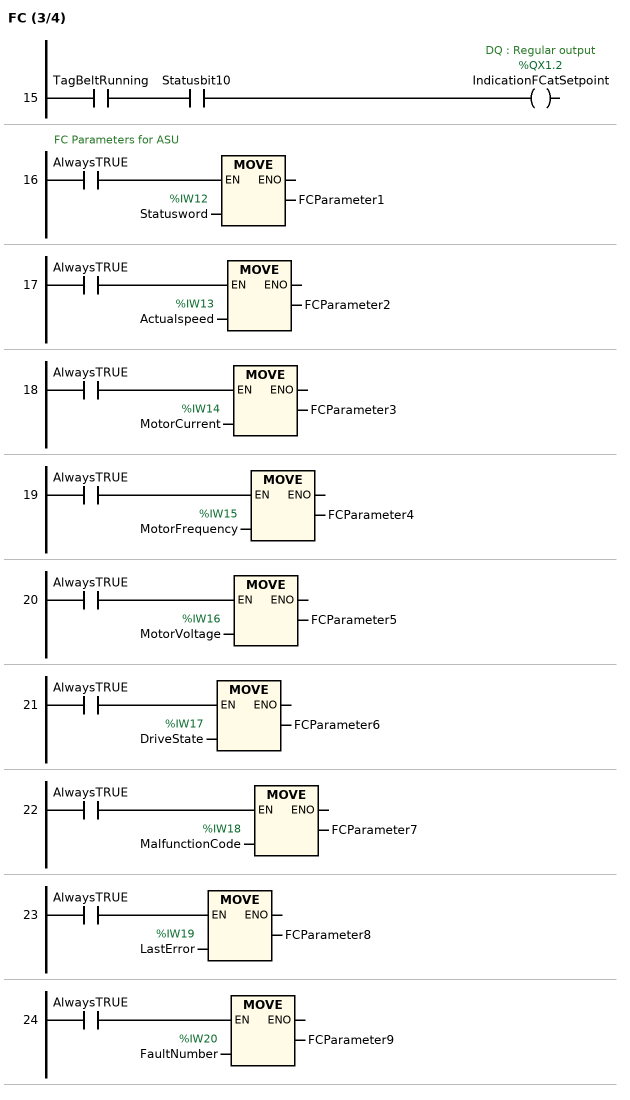
// NETWORK 15
//   IndicationFCatSetpoint: DQ : Regular output | AT %QX1.2
IndicationFCatSetpoint := TagBeltRunning AND Statusbit10;

// NETWORK 16
// FC Parameters for ASU
//   Statusword: ATV340_1 : ETA Status word | AT %IW12
//   FCParameter1: AT %MW32
IF AlwaysTRUE THEN FCParameter1 := Statusword; END_IF

// NETWORK 17
//   Actualspeed: ATV340_1 : Output speed | AT %IW13
//   FCParameter2: AT %MW33
IF AlwaysTRUE THEN FCParameter2 := Actualspeed; END_IF

// NETWORK 18
//   MotorCurrent: ATV340_1 : bom | AT %IW14
//   FCParameter3: AT %MW34
IF AlwaysTRUE THEN FCParameter3 := MotorCurrent; END_IF

// NETWORK 19
//   MotorFrequency: ATV340_1 : configurable | AT %IW15
//   FCParameter4: AT %MW35
IF AlwaysTRUE THEN FCParameter4 := MotorFrequency; END_IF

// NETWORK 20
//   MotorVoltage: ATV340_1 : configurable | AT %IW16
//   FCParameter5: AT %MW36
IF AlwaysTRUE THEN FCParameter5 := MotorVoltage; END_IF

// NETWORK 21
//   DriveState: ATV340_1 : configurable | AT %IW17
//   FCParameter6: AT %MW37
IF AlwaysTRUE THEN FCParameter6 := DriveState; END_IF

// NETWORK 22
//   MalfunctionCode: ATV340_1 : configurable | AT %IW18
//   FCParameter7: AT %MW38
IF AlwaysTRUE THEN FCParameter7 := MalfunctionCode; END_IF

// NETWORK 23
//   LastError: ATV340_1 : configurable | AT %IW19
//   FCParameter8: AT %MW39
IF AlwaysTRUE THEN FCParameter8 := LastError; END_IF

// NETWORK 24
//   FaultNumber: ATV340_1 : configurable | AT %IW20
//   FCParameter9: AT %MW40
IF AlwaysTRUE THEN FCParameter9 := FaultNumber; END_IF

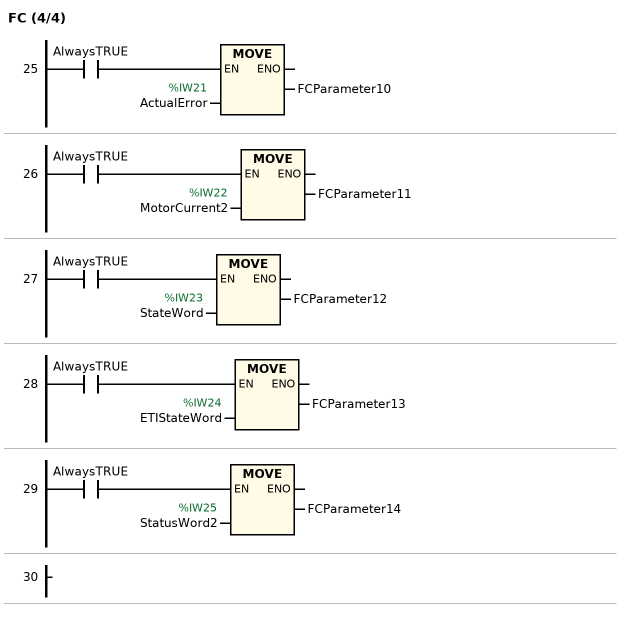
// NETWORK 25
//   ActualError: ATV340_1 : configurable | AT %IW21
//   FCParameter10: AT %MW41
IF AlwaysTRUE THEN FCParameter10 := ActualError; END_IF

// NETWORK 26
//   MotorCurrent2: ATV340_1 : configurable | AT %IW22
//   FCParameter11: AT %MW42
IF AlwaysTRUE THEN FCParameter11 := MotorCurrent2; END_IF

// NETWORK 27
//   StateWord: ATV340_1 : configurable | AT %IW23
//   FCParameter12: AT %MW43
IF AlwaysTRUE THEN FCParameter12 := StateWord; END_IF

// NETWORK 28
//   ETIStateWord: ATV340_1 : configurable | AT %IW24
//   FCParameter13: AT %MW44
IF AlwaysTRUE THEN FCParameter13 := ETIStateWord; END_IF

// NETWORK 29
//   StatusWord2: ATV340_1 : configurable | AT %IW25
//   FCParameter14: AT %MW45
IF AlwaysTRUE THEN FCParameter14 := StatusWord2; END_IF

// NETWORK 30

END_PROGRAM

// MyController/Application/Encoder
PROGRAM Encoder
VAR
	EXPERTSetParam_0: EXPERTSetParam;
	TriggerSetNewPresetFront: BOOL;
	TriggerSetNewPresetEnd: BOOL;
	TriggerSetNewPresetPLCRestart: BOOL;
	testBool2: BOOL;
	testHSCRef: EXPERT_REF;
	ReadDone: BOOL;
	ReadBusy: BOOL;
	ReadError: BOOL;
	ReadErrorID: EXPERT_ERR_TYPE;
	ExpertSetParamCache: DINT;
	ParamValueRead: DINT;
	
	PresetBusy: BOOL; 
	PresetError: BOOL; 
	PresetErrID: EXPERT_ERR_TYPE; 
	EXPERTGetParam_0: EXPERTGetParam;
	TriggerSetNewPreset: BOOL;
	ColdStartSignalFilter: TON;
	TONColdStartSignalFilterService: TIME;
	
	TONFrontEndPositionEncoderFilter: TON;
	TONRearEndPositionEncoderFilter: TON;
	TONFrontEndPositionEncoderFilterService: TIME;
	TONRearEndPositionEncoderFilterService: TIME;
END_VAR
VAR // added by the converter: edge detectors and wires of the graphical bodies
    _w1, _w2, _w3, _w4 : BOOL;
    _rt1 : R_TRIG;
END_VAR

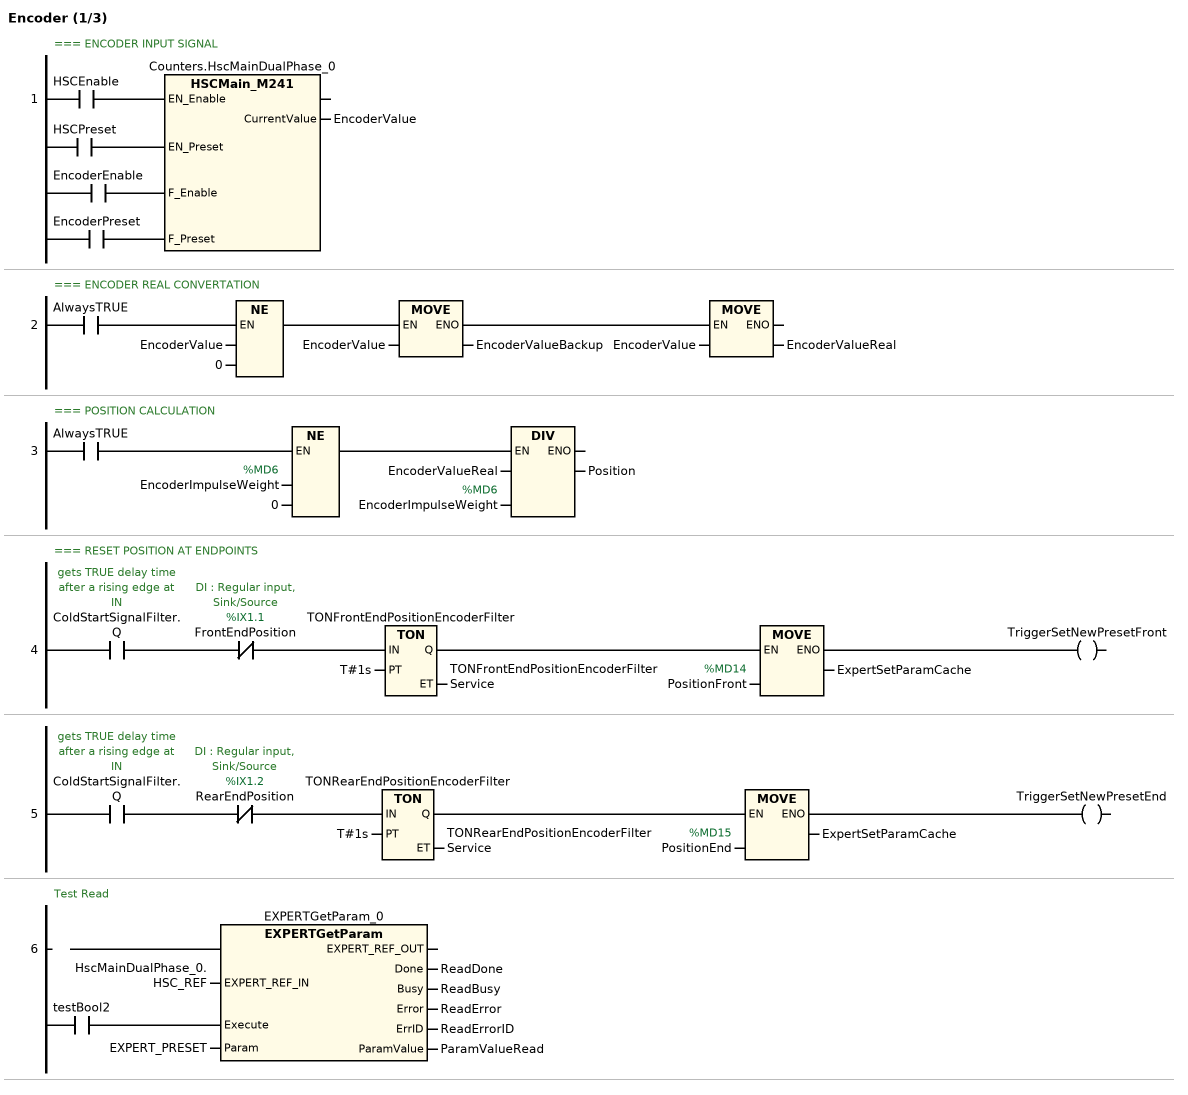
// NETWORK 1
// === ENCODER INPUT SIGNAL
Counters.HscMainDualPhase_0(
    EN_Enable := HSCEnable,
    EN_Preset := HSCPreset,
    F_Enable := EncoderEnable,
    F_Preset := EncoderPreset,
    CurrentValue => EncoderValue); // HSCMain_M241

// NETWORK 2
// === ENCODER REAL CONVERTATION
_w1 := AlwaysTRUE AND EncoderValue <> 0;
IF _w1 THEN EncoderValueBackup := EncoderValue; END_IF
IF _w1 THEN EncoderValueReal := EncoderValue; END_IF

// NETWORK 3
// === POSITION CALCULATION
//   EncoderImpulseWeight: AT %MD6
//   Position: AT %MD13
IF AlwaysTRUE AND EncoderImpulseWeight <> 0 THEN Position := EncoderValueReal / EncoderImpulseWeight; END_IF

// NETWORK 4
// === RESET POSITION AT ENDPOINTS
//   ColdStartSignalFilter.Q: gets TRUE delay time after a rising edge at IN
//   FrontEndPosition: DI : Regular input, Sink/Source | AT %IX1.1
//   PositionFront: AT %MD14
TONFrontEndPositionEncoderFilter(
    IN := ColdStartSignalFilter.Q AND NOT FrontEndPosition,
    PT := T#1s,
    ET => TONFrontEndPositionEncoderFilterService); // TON
_w2 := TONFrontEndPositionEncoderFilter.Q;
IF _w2 THEN ExpertSetParamCache := PositionFront; END_IF
TriggerSetNewPresetFront := _w2;

// NETWORK 5
//   ColdStartSignalFilter.Q: gets TRUE delay time after a rising edge at IN
//   RearEndPosition: DI : Regular input, Sink/Source | AT %IX1.2
//   PositionEnd: AT %MD15
TONRearEndPositionEncoderFilter(
    IN := ColdStartSignalFilter.Q AND NOT RearEndPosition,
    PT := T#1s,
    ET => TONRearEndPositionEncoderFilterService); // TON
_w3 := TONRearEndPositionEncoderFilter.Q;
IF _w3 THEN ExpertSetParamCache := PositionEnd; END_IF
TriggerSetNewPresetEnd := _w3;

// NETWORK 6
// Test Read
//   HscMainDualPhase_0.HSC_REF: Reference to the HSC. To be used as input of administrative Function block.
EXPERTGetParam_0(
    EXPERT_REF_IN := HscMainDualPhase_0.HSC_REF,
    Execute := testBool2,
    Param := EXPERT_PRESET,
    Done => ReadDone,
    Busy => ReadBusy,
    Error => ReadError,
    ErrID => ReadErrorID,
    ParamValue => ParamValueRead); // EXPERTGetParam

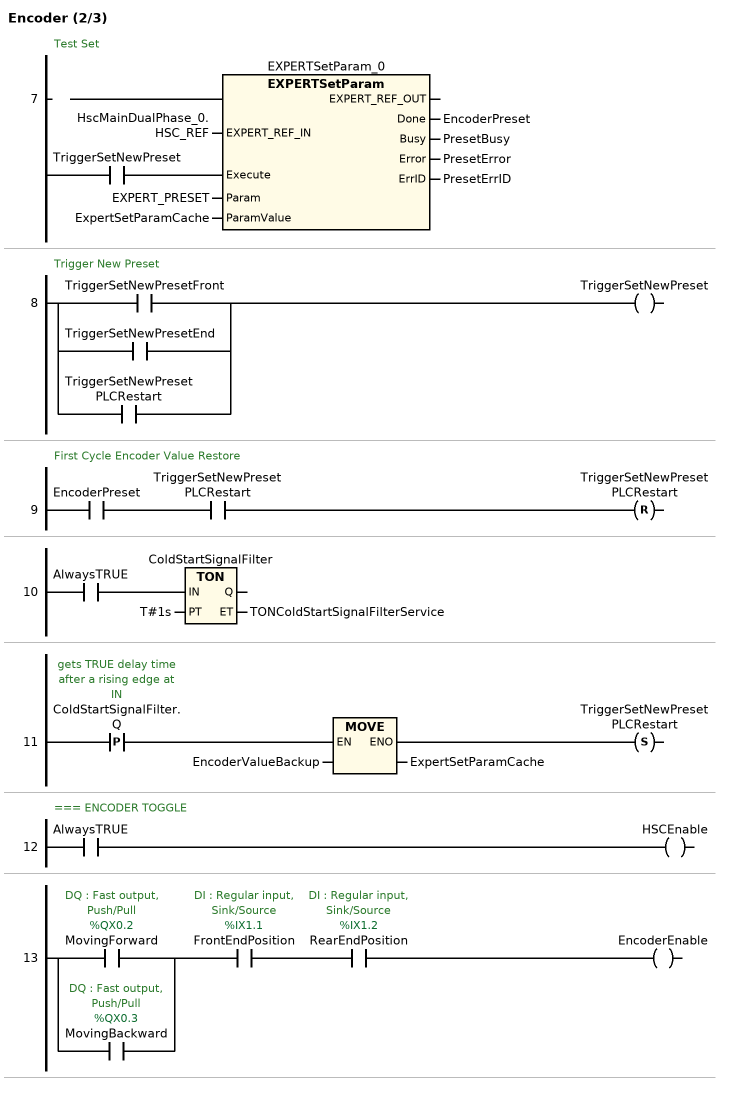
// NETWORK 7
// Test Set
//   HscMainDualPhase_0.HSC_REF: Reference to the HSC. To be used as input of administrative Function block.
EXPERTSetParam_0(
    EXPERT_REF_IN := HscMainDualPhase_0.HSC_REF,
    Execute := TriggerSetNewPreset,
    Param := EXPERT_PRESET,
    ParamValue := ExpertSetParamCache,
    Done => EncoderPreset,
    Busy => PresetBusy,
    Error => PresetError,
    ErrID => PresetErrID); // EXPERTSetParam

// NETWORK 8
// Trigger New Preset
TriggerSetNewPreset := TriggerSetNewPresetFront OR TriggerSetNewPresetEnd OR TriggerSetNewPresetPLCRestart;

// NETWORK 9
// First Cycle Encoder Value Restore
TriggerSetNewPresetPLCRestart R= EncoderPreset AND TriggerSetNewPresetPLCRestart;

// NETWORK 10
ColdStartSignalFilter(IN := AlwaysTRUE, PT := T#1s, ET => TONColdStartSignalFilterService); // TON

// NETWORK 11
//   ColdStartSignalFilter.Q: gets TRUE delay time after a rising edge at IN
_rt1(CLK := ColdStartSignalFilter.Q);
_w4 := _rt1.Q;
IF _w4 THEN ExpertSetParamCache := EncoderValueBackup; END_IF
TriggerSetNewPresetPLCRestart S= _w4;

// NETWORK 12
// === ENCODER TOGGLE
HSCEnable := AlwaysTRUE;

// NETWORK 13
//   MovingForward: DQ : Fast output, Push/Pull | AT %QX0.2
//   MovingBackward: DQ : Fast output, Push/Pull | AT %QX0.3
//   FrontEndPosition: DI : Regular input, Sink/Source | AT %IX1.1
//   RearEndPosition: DI : Regular input, Sink/Source | AT %IX1.2
EncoderEnable := (MovingForward OR MovingBackward) AND FrontEndPosition AND RearEndPosition;

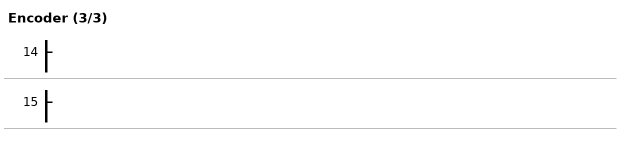
// NETWORK 14

// NETWORK 15

END_PROGRAM

// MyController/Application/LevelSensors
PROGRAM LevelSensors
VAR
	LIN_TRAFO_0: LIN_TRAFO;
	LIN_TRAFO_1: LIN_TRAFO;
END_VAR

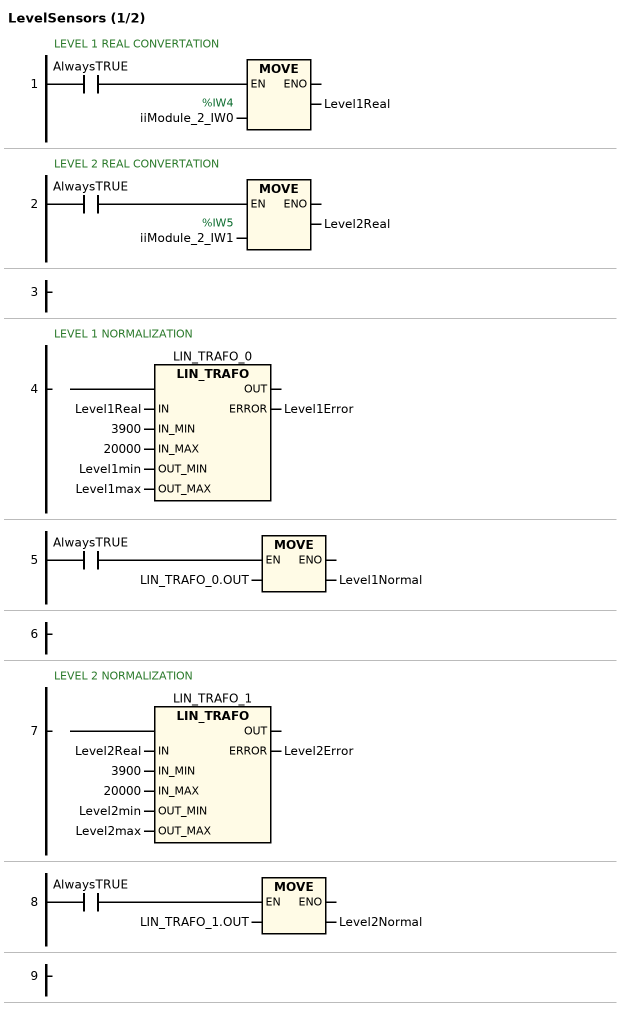
// NETWORK 1
// LEVEL 1 REAL CONVERTATION
//   iiModule_2_IW0: Module_2 : LevelSensor1 | AT %IW4
IF AlwaysTRUE THEN Level1Real := iiModule_2_IW0; END_IF

// NETWORK 2
// LEVEL 2 REAL CONVERTATION
//   iiModule_2_IW1: Module_2 : LevelSensor2 | AT %IW5
IF AlwaysTRUE THEN Level2Real := iiModule_2_IW1; END_IF

// NETWORK 3

// NETWORK 4
// LEVEL 1 NORMALIZATION
LIN_TRAFO_0(
    IN := Level1Real,
    IN_MIN := 3900,
    IN_MAX := 20000,
    OUT_MIN := Level1min,
    OUT_MAX := Level1max,
    ERROR => Level1Error); // LIN_TRAFO

// NETWORK 5
//   LIN_TRAFO_0.OUT: output value
IF AlwaysTRUE THEN Level1Normal := LIN_TRAFO_0.OUT; END_IF

// NETWORK 6

// NETWORK 7
// LEVEL 2 NORMALIZATION
LIN_TRAFO_1(
    IN := Level2Real,
    IN_MIN := 3900,
    IN_MAX := 20000,
    OUT_MIN := Level2min,
    OUT_MAX := Level2max,
    ERROR => Level2Error); // LIN_TRAFO

// NETWORK 8
//   LIN_TRAFO_1.OUT: output value
IF AlwaysTRUE THEN Level2Normal := LIN_TRAFO_1.OUT; END_IF

// NETWORK 9

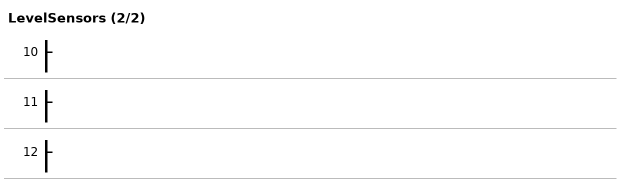
// NETWORK 10

// NETWORK 11

// NETWORK 12

END_PROGRAM

// MyController/Application/HMI
PROGRAM HMI
VAR
END_VAR

